            state1.dvar_M_HardwareMapDH_out_a_x2testing := TRUE;
            state1.dvar_M_HardwareMapDH := elit_init3;

            state0 := state1;
        END_IF;
    END_IF;

    // Event "tau".
    IF NOT progress THEN
        IF (state0.dvar_M_HardwareMapDH) = (elit_init3) THEN
            progress := TRUE;
            state1 := state0;

            state1.dvar_M_HardwareMapDH_out_a_transfer2pickpos := TRUE;
            state1.dvar_M_HardwareMapDH := elit_init4;

            state0 := state1;
        END_IF;
    END_IF;

    // Event "tau".
    IF NOT progress THEN
        b1 := (state0.dvar_M_HardwareMapDH) = (elit_init4);
        b1 := b1 AND (ivar_s_transfer_atpickup);
        IF b1 THEN
            progress := TRUE;
            state1 := state0;

            state1.dvar_M_HardwareMapDH_out_a_transfer2pickpos := FALSE;
            state1.dvar_M_HardwareMapDH := elit_init5;

            state0 := state1;
        END_IF;
    END_IF;

    // Event "tau".
    IF NOT progress THEN
        IF (state0.dvar_M_HardwareMapDH) = (elit_init5) THEN
            progress := TRUE;
            state1 := state0;

            state1.dvar_M_HardwareMapDH_out_a_transfer2droppos := TRUE;
            state1.dvar_M_HardwareMapDH := elit_init6;

            state0 := state1;
        END_IF;
    END_IF;

    // Event "tau".
    IF NOT progress THEN
        b1 := (state0.dvar_M_HardwareMapDH) = (elit_init6);
        b1 := b1 AND (ivar_s_transfer_athalfway);
        IF b1 THEN
            progress := TRUE;
            state1 := state0;

            state1.dvar_M_HardwareMapDH_out_a_transfer2droppos := FALSE;
            state1.dvar_M_HardwareMapDH := elit_init7;

            state0 := state1;
        END_IF;
    END_IF;

    // Event "tau".
    IF NOT progress THEN
        IF (state0.dvar_M_HardwareMapDH) = (elit_init7) THEN
            progress := TRUE;
            state1 := state0;

            state1.dvar_M_HardwareMapDH_out_a_x2distributing := FALSE;
            state1.dvar_M_HardwareMapDH := elit_init8;

            state0 := state1;
        END_IF;
    END_IF;

    // Event "tau".
    IF NOT progress THEN
        b1 := (state0.dvar_M_HardwareMapDH) = (elit_init8);
        b1 := b1 AND (ivar_s_xpos_atdrop);
        IF b1 THEN
            progress := TRUE;
            state1 := state0;

            state1.dvar_M_HardwareMapDH_out_a_x2distributing := TRUE;
            state1.cvar_M_HardwareMapDH_t := 0.0;
            state1.dvar_M_HardwareMapDH := elit_init9;

            state0 := state1;
        END_IF;
    END_IF;

    // Event "tau".
    IF NOT progress THEN
        b1 := (state0.dvar_M_HardwareMapDH) = (elit_init9);
        b1 := b1 AND ((state0.cvar_M_HardwareMapDH_t) >= (1));
        IF b1 THEN
            progress := TRUE;
            state1 := state0;

            state1.dvar_M_HardwareMapDH := elit_init_sensor_check;

            state0 := state1;
        END_IF;
    END_IF;

    // Event "tau".
    IF NOT progress THEN
        b1 := (state0.dvar_M_HardwareMapDH) = (elit_init_sensor_check);
        b1 := b1 AND (ivar_s_Dstartbutton);
        IF b1 THEN
            progress := TRUE;
            state1 := state0;

            state1.dvar_M_HardwareMapDH_init_err_sen_idx := 0;
            state1.dvar_M_HardwareMapDH := elit_init_error;

            state0 := state1;
        END_IF;
    END_IF;

    // Event "tau".
    IF NOT progress THEN
        b1 := (state0.dvar_M_HardwareMapDH) = (elit_init_sensor_check);
        b1 := b1 AND (NOT(ivar_s_Dstopbutton));
        IF b1 THEN
            progress := TRUE;
            state1 := state0;

            state1.dvar_M_HardwareMapDH_init_err_sen_idx := 1;
            state1.dvar_M_HardwareMapDH := elit_init_error;

            state0 := state1;
        END_IF;
    END_IF;

    // Event "tau".
    IF NOT progress THEN
        b1 := (state0.dvar_M_HardwareMapDH) = (elit_init_sensor_check);
        b1 := b1 AND (ivar_s_Dautoswitch);
        IF b1 THEN
            progress := TRUE;
            state1 := state0;

            state1.dvar_M_HardwareMapDH_init_err_sen_idx := 2;
            state1.dvar_M_HardwareMapDH := elit_init_error;

            state0 := state1;
        END_IF;
    END_IF;

    // Event "tau".
    IF NOT progress THEN
        b1 := (state0.dvar_M_HardwareMapDH) = (elit_init_sensor_check);
        b1 := b1 AND (ivar_s_Dresetbutton);
        IF b1 THEN
            progress := TRUE;
            state1 := state0;

            state1.dvar_M_HardwareMapDH_init_err_sen_idx := 3;
            state1.dvar_M_HardwareMapDH := elit_init_error;

            state0 := state1;
        END_IF;
    END_IF;

    // Event "tau".
    IF NOT progress THEN
        b1 := (state0.dvar_M_HardwareMapDH) = (elit_init_sensor_check);
        b1 := b1 AND (ivar_s_Din4);
        IF b1 THEN
            progress := TRUE;
            state1 := state0;

            state1.dvar_M_HardwareMapDH_init_err_sen_idx := 4;
            state1.dvar_M_HardwareMapDH := elit_init_error;

            state0 := state1;
        END_IF;
    END_IF;

    // Event "tau".
    IF NOT progress THEN
        b1 := (state0.dvar_M_HardwareMapDH) = (elit_init_sensor_check);
        b1 := b1 AND (ivar_s_Din5);
        IF b1 THEN
            progress := TRUE;
            state1 := state0;

            state1.dvar_M_HardwareMapDH_init_err_sen_idx := 5;
            state1.dvar_M_HardwareMapDH := elit_init_error;

            state0 := state1;
        END_IF;
    END_IF;

    // Event "tau".
    IF NOT progress THEN
        b1 := (state0.dvar_M_HardwareMapDH) = (elit_init_sensor_check);
        b1 := b1 AND (ivar_s_Din6);
        IF b1 THEN
            progress := TRUE;
            state1 := state0;

            state1.dvar_M_HardwareMapDH_init_err_sen_idx := 6;
            state1.dvar_M_HardwareMapDH := elit_init_error;

            state0 := state1;
        END_IF;
    END_IF;

    // Event "tau".
    IF NOT progress THEN
        b1 := (state0.dvar_M_HardwareMapDH) = (elit_init_sensor_check);
        b1 := b1 AND (ivar_s_Din7);
        IF b1 THEN
            progress := TRUE;
            state1 := state0;

            state1.dvar_M_HardwareMapDH_init_err_sen_idx := 7;
            state1.dvar_M_HardwareMapDH := elit_init_error;

            state0 := state1;
        END_IF;
    END_IF;

    // Event "tau".
    IF NOT progress THEN
        b1 := (state0.dvar_M_HardwareMapDH) = (elit_init_sensor_check);
        b1 := b1 AND (NOT(ivar_s_pusher1_in));
        IF b1 THEN
            progress := TRUE;
            state1 := state0;

            state1.dvar_M_HardwareMapDH_init_err_sen_idx := 8;
            state1.dvar_M_HardwareMapDH := elit_init_error;

            state0 := state1;
        END_IF;
    END_IF;

    // Event "tau".
    IF NOT progress THEN
        b1 := (state0.dvar_M_HardwareMapDH) = (elit_init_sensor_check);
        b1 := b1 AND (ivar_s_pusher1_out);
        IF b1 THEN
            progress := TRUE;
            state1 := state0;

            state1.dvar_M_HardwareMapDH_init_err_sen_idx := 9;
            state1.dvar_M_HardwareMapDH := elit_init_error;

            state0 := state1;
        END_IF;
    END_IF;

    // Event "tau".
    IF NOT progress THEN
        b1 := (state0.dvar_M_HardwareMapDH) = (elit_init_sensor_check);
        b1 := b1 AND (NOT(ivar_s_stack1filled));
        IF b1 THEN
            progress := TRUE;
            state1 := state0;

            state1.dvar_M_HardwareMapDH_init_err_sen_idx := 10;
            state1.dvar_M_HardwareMapDH := elit_init_error;

            state0 := state1;
        END_IF;
    END_IF;

    // Event "tau".
    IF NOT progress THEN
        b1 := (state0.dvar_M_HardwareMapDH) = (elit_init_sensor_check);
        b1 := b1 AND (ivar_s_product1);
        IF b1 THEN
            progress := TRUE;
            state1 := state0;

            state1.dvar_M_HardwareMapDH_init_err_sen_idx := 11;
            state1.dvar_M_HardwareMapDH := elit_init_error;

            state0 := state1;
        END_IF;
    END_IF;

    // Event "tau".
    IF NOT progress THEN
        b1 := (state0.dvar_M_HardwareMapDH) = (elit_init_sensor_check);
        b1 := b1 AND (NOT(ivar_s_pusher2_in));
        IF b1 THEN
            progress := TRUE;
            state1 := state0;

            state1.dvar_M_HardwareMapDH_init_err_sen_idx := 12;
            state1.dvar_M_HardwareMapDH := elit_init_error;

            state0 := state1;
        END_IF;
    END_IF;

    // Event "tau".
    IF NOT progress THEN
        b1 := (state0.dvar_M_HardwareMapDH) = (elit_init_sensor_check);
        b1 := b1 AND (ivar_s_pusher2_out);
        IF b1 THEN
            progress := TRUE;
            state1 := state0;

            state1.dvar_M_HardwareMapDH_init_err_sen_idx := 13;
            state1.dvar_M_HardwareMapDH := elit_init_error;

            state0 := state1;
        END_IF;
    END_IF;

    // Event "tau".
    IF NOT progress THEN
        b1 := (state0.dvar_M_HardwareMapDH) = (elit_init_sensor_check);
        b1 := b1 AND (NOT(ivar_s_stack2filled));
        IF b1 THEN
            progress := TRUE;
            state1 := state0;

            state1.dvar_M_HardwareMapDH_init_err_sen_idx := 14;
            state1.dvar_M_HardwareMapDH := elit_init_error;

            state0 := state1;
        END_IF;
    END_IF;

    // Event "tau".
    IF NOT progress THEN
        b1 := (state0.dvar_M_HardwareMapDH) = (elit_init_sensor_check);
        b1 := b1 AND (ivar_s_product2);
        IF b1 THEN
            progress := TRUE;
            state1 := state0;

            state1.dvar_M_HardwareMapDH_init_err_sen_idx := 15;
            state1.dvar_M_HardwareMapDH := elit_init_error;

            state0 := state1;
        END_IF;
    END_IF;

    // Event "tau".
    IF NOT progress THEN
        b1 := (state0.dvar_M_HardwareMapDH) = (elit_init_sensor_check);
        b1 := b1 AND (NOT(ivar_s_pusher3_in));
        IF b1 THEN
            progress := TRUE;
            state1 := state0;

            state1.dvar_M_HardwareMapDH_init_err_sen_idx := 16;
            state1.dvar_M_HardwareMapDH := elit_init_error;

            state0 := state1;
        END_IF;
    END_IF;

    // Event "tau".
    IF NOT progress THEN
        b1 := (state0.dvar_M_HardwareMapDH) = (elit_init_sensor_check);
        b1 := b1 AND (ivar_s_pusher3_out);
        IF b1 THEN
            progress := TRUE;
            state1 := state0;

            state1.dvar_M_HardwareMapDH_init_err_sen_idx := 17;
            state1.dvar_M_HardwareMapDH := elit_init_error;

            state0 := state1;
        END_IF;
    END_IF;

    // Event "tau".
    IF NOT progress THEN
        b1 := (state0.dvar_M_HardwareMapDH) = (elit_init_sensor_check);
        b1 := b1 AND (NOT(ivar_s_stack3filled));
        IF b1 THEN
            progress := TRUE;
            state1 := state0;

            state1.dvar_M_HardwareMapDH_init_err_sen_idx := 18;
            state1.dvar_M_HardwareMapDH := elit_init_error;

            state0 := state1;
        END_IF;
    END_IF;

    // Event "tau".
    IF NOT progress THEN
        b1 := (state0.dvar_M_HardwareMapDH) = (elit_init_sensor_check);
        b1 := b1 AND (ivar_s_product3);
        IF b1 THEN
            progress := TRUE;
            state1 := state0;

            state1.dvar_M_HardwareMapDH_init_err_sen_idx := 19;
            state1.dvar_M_HardwareMapDH := elit_init_error;

            state0 := state1;
        END_IF;
    END_IF;

    // Event "tau".
    IF NOT progress THEN
        b1 := (state0.dvar_M_HardwareMapDH) = (elit_init_sensor_check);
        b1 := b1 AND (ivar_s_Hstartbutton);
        IF b1 THEN
            progress := TRUE;
            state1 := state0;

            state1.dvar_M_HardwareMapDH_init_err_sen_idx := 22;
            state1.dvar_M_HardwareMapDH := elit_init_error;

            state0 := state1;
        END_IF;
    END_IF;

    // Event "tau".
    IF NOT progress THEN
        b1 := (state0.dvar_M_HardwareMapDH) = (elit_init_sensor_check);
        b1 := b1 AND (NOT(ivar_s_Hstopbutton));
        IF b1 THEN
            progress := TRUE;
            state1 := state0;

            state1.dvar_M_HardwareMapDH_init_err_sen_idx := 23;
            state1.dvar_M_HardwareMapDH := elit_init_error;

            state0 := state1;
        END_IF;
    END_IF;

    // Event "tau".
    IF NOT progress THEN
        b1 := (state0.dvar_M_HardwareMapDH) = (elit_init_sensor_check);
        b1 := b1 AND (ivar_s_Hautoswitch);
        IF b1 THEN
            progress := TRUE;
            state1 := state0;

            state1.dvar_M_HardwareMapDH_init_err_sen_idx := 24;
            state1.dvar_M_HardwareMapDH := elit_init_error;

            state0 := state1;
        END_IF;
    END_IF;

    // Event "tau".
    IF NOT progress THEN
        b1 := (state0.dvar_M_HardwareMapDH) = (elit_init_sensor_check);
        b1 := b1 AND (ivar_s_Hresetbutton);
        IF b1 THEN
            progress := TRUE;
            state1 := state0;

            state1.dvar_M_HardwareMapDH_init_err_sen_idx := 25;
            state1.dvar_M_HardwareMapDH := elit_init_error;

            state0 := state1;
        END_IF;
    END_IF;

    // Event "tau".
    IF NOT progress THEN
        b1 := (state0.dvar_M_HardwareMapDH) = (elit_init_sensor_check);
        b1 := b1 AND (ivar_s_Hin4);
        IF b1 THEN
            progress := TRUE;
            state1 := state0;

            state1.dvar_M_HardwareMapDH_init_err_sen_idx := 26;
            state1.dvar_M_HardwareMapDH := elit_init_error;

            state0 := state1;
        END_IF;
    END_IF;

    // Event "tau".
    IF NOT progress THEN
        b1 := (state0.dvar_M_HardwareMapDH) = (elit_init_sensor_check);
        b1 := b1 AND (ivar_s_Hin5);
        IF b1 THEN
            progress := TRUE;
            state1 := state0;

            state1.dvar_M_HardwareMapDH_init_err_sen_idx := 27;
            state1.dvar_M_HardwareMapDH := elit_init_error;

            state0 := state1;
        END_IF;
    END_IF;

    // Event "tau".
    IF NOT progress THEN
        b1 := (state0.dvar_M_HardwareMapDH) = (elit_init_sensor_check);
        b1 := b1 AND (ivar_s_Hin6);
        IF b1 THEN
            progress := TRUE;
            state1 := state0;

            state1.dvar_M_HardwareMapDH_init_err_sen_idx := 28;
            state1.dvar_M_HardwareMapDH := elit_init_error;

            state0 := state1;
        END_IF;
    END_IF;

    // Event "tau".
    IF NOT progress THEN
        b1 := (state0.dvar_M_HardwareMapDH) = (elit_init_sensor_check);
        b1 := b1 AND (ivar_s_Hin7);
        IF b1 THEN
            progress := TRUE;
            state1 := state0;

            state1.dvar_M_HardwareMapDH_init_err_sen_idx := 29;
            state1.dvar_M_HardwareMapDH := elit_init_error;

            state0 := state1;
        END_IF;
    END_IF;

    // Event "tau".
    IF NOT progress THEN
        b1 := (state0.dvar_M_HardwareMapDH) = (elit_init_sensor_check);
        b1 := b1 AND (ivar_s_xpos_at1);
        IF b1 THEN
            progress := TRUE;
            state1 := state0;

            state1.dvar_M_HardwareMapDH_init_err_sen_idx := 33;
            state1.dvar_M_HardwareMapDH := elit_init_error;

            state0 := state1;
        END_IF;
    END_IF;

    // Event "tau".
    IF NOT progress THEN
        b1 := (state0.dvar_M_HardwareMapDH) = (elit_init_sensor_check);
        b1 := b1 AND (ivar_s_xpos_at2);
        IF b1 THEN
            progress := TRUE;
            state1 := state0;

            state1.dvar_M_HardwareMapDH_init_err_sen_idx := 34;
            state1.dvar_M_HardwareMapDH := elit_init_error;

            state0 := state1;
        END_IF;
    END_IF;

    // Event "tau".
    IF NOT progress THEN
        b1 := (state0.dvar_M_HardwareMapDH) = (elit_init_sensor_check);
        b1 := b1 AND (ivar_s_xpos_at3);
        IF b1 THEN
            progress := TRUE;
            state1 := state0;

            state1.dvar_M_HardwareMapDH_init_err_sen_idx := 35;
            state1.dvar_M_HardwareMapDH := elit_init_error;

            state0 := state1;
        END_IF;
    END_IF;

    // Event "tau".
    IF NOT progress THEN
        b1 := (state0.dvar_M_HardwareMapDH) = (elit_init_sensor_check);
        b1 := b1 AND (NOT(ivar_s_xpos_atdrop));
        IF b1 THEN
            progress := TRUE;
            state1 := state0;

            state1.dvar_M_HardwareMapDH_init_err_sen_idx := 36;
            state1.dvar_M_HardwareMapDH := elit_init_error;

            state0 := state1;
        END_IF;
    END_IF;

    // Event "tau".
    IF NOT progress THEN
        b1 := (state0.dvar_M_HardwareMapDH) = (elit_init_sensor_check);
        b1 := b1 AND (NOT(ivar_s_zpos_atup));
        IF b1 THEN
            progress := TRUE;
            state1 := state0;

            state1.dvar_M_HardwareMapDH_init_err_sen_idx := 37;
            state1.dvar_M_HardwareMapDH := elit_init_error;

            state0 := state1;
        END_IF;
    END_IF;

    // Event "tau".
    IF NOT progress THEN
        b1 := (state0.dvar_M_HardwareMapDH) = (elit_init_sensor_check);
        b1 := b1 AND (ivar_s_zpos_atdown);
        IF b1 THEN
            progress := TRUE;
            state1 := state0;

            state1.dvar_M_HardwareMapDH_init_err_sen_idx := 38;
            state1.dvar_M_HardwareMapDH := elit_init_error;

            state0 := state1;
        END_IF;
    END_IF;

    // Event "tau".
    IF NOT progress THEN
        b1 := (state0.dvar_M_HardwareMapDH) = (elit_init_sensor_check);
        b1 := b1 AND (ivar_s_gripper);
        IF b1 THEN
            progress := TRUE;
            state1 := state0;

            state1.dvar_M_HardwareMapDH_init_err_sen_idx := 39;
            state1.dvar_M_HardwareMapDH := elit_init_error;

            state0 := state1;
        END_IF;
    END_IF;

    // Event "tau".
    IF NOT progress THEN
        b1 := (state0.dvar_M_HardwareMapDH) = (elit_init_sensor_check);
        b1 := b1 AND (ivar_s_transfer_atpickup);
        IF b1 THEN
            progress := TRUE;
            state1 := state0;

            state1.dvar_M_HardwareMapDH_init_err_sen_idx := 40;
            state1.dvar_M_HardwareMapDH := elit_init_error;

            state0 := state1;
        END_IF;
    END_IF;

    // Event "tau".
    IF NOT progress THEN
        b1 := (state0.dvar_M_HardwareMapDH) = (elit_init_sensor_check);
        b1 := b1 AND (ivar_s_transfer_atdrop);
        IF b1 THEN
            progress := TRUE;
            state1 := state0;

            state1.dvar_M_HardwareMapDH_init_err_sen_idx := 41;
            state1.dvar_M_HardwareMapDH := elit_init_error;

            state0 := state1;
        END_IF;
    END_IF;

    // Event "tau".
    IF NOT progress THEN
        b1 := (state0.dvar_M_HardwareMapDH) = (elit_init_sensor_check);
        b1 := b1 AND (NOT(ivar_s_transfer_athalfway));
        IF b1 THEN
            progress := TRUE;
            state1 := state0;

            state1.dvar_M_HardwareMapDH_init_err_sen_idx := 42;
            state1.dvar_M_HardwareMapDH := elit_init_error;

            state0 := state1;
        END_IF;
    END_IF;

    // Event "tau".
    IF NOT progress THEN
        b1 := (state0.dvar_M_HardwareMapDH) = (elit_init_sensor_check);
        b1 := b1 AND (ivar_s_vacuum);
        IF b1 THEN
            progress := TRUE;
            state1 := state0;

            state1.dvar_M_HardwareMapDH_init_err_sen_idx := 43;
            state1.dvar_M_HardwareMapDH := elit_init_error;

            state0 := state1;
        END_IF;
    END_IF;

    // Event "tau".
    IF NOT progress THEN
        b1 := (state0.dvar_M_HardwareMapDH) = (elit_init_sensor_check);
        b1 := b1 AND (ivar_s_product4);
        IF b1 THEN
            progress := TRUE;
            state1 := state0;

            state1.dvar_M_HardwareMapDH_init_err_sen_idx := 44;
            state1.dvar_M_HardwareMapDH := elit_init_error;

            state0 := state1;
        END_IF;
    END_IF;

    // Event "tau".
    IF NOT progress THEN
        b1 := (state0.dvar_M_HardwareMapDH) = (elit_init_sensor_check);
        b1 := b1 AND (NOT(ivar_s_Dstartbutton));
        b1 := b1 AND (ivar_s_Dstopbutton);
        b1 := b1 AND (NOT(ivar_s_Dautoswitch));
        b1 := b1 AND (NOT(ivar_s_Dresetbutton));
        b1 := b1 AND (NOT(ivar_s_Din4));
        b1 := b1 AND (NOT(ivar_s_Din5));
        b1 := b1 AND (NOT(ivar_s_Din6));
        b1 := b1 AND (NOT(ivar_s_Din7));
        b1 := b1 AND (ivar_s_pusher1_in);
        b1 := b1 AND (NOT(ivar_s_pusher1_out));
        b1 := b1 AND (ivar_s_stack1filled);
        b1 := b1 AND (NOT(ivar_s_product1));
        b1 := b1 AND (ivar_s_pusher2_in);
        b1 := b1 AND (NOT(ivar_s_pusher2_out));
        b1 := b1 AND (ivar_s_stack2filled);
        b1 := b1 AND (NOT(ivar_s_product2));
        b1 := b1 AND (ivar_s_pusher3_in);
        b1 := b1 AND (NOT(ivar_s_pusher3_out));
        b1 := b1 AND (ivar_s_stack3filled);
        b1 := b1 AND (NOT(ivar_s_product3));
        b1 := b1 AND (NOT(ivar_s_Hstartbutton));
        b1 := b1 AND (ivar_s_Hstopbutton);
        b1 := b1 AND (NOT(ivar_s_Hautoswitch));
        b1 := b1 AND (NOT(ivar_s_Hresetbutton));
        b1 := b1 AND (NOT(ivar_s_Hin4));
        b1 := b1 AND (NOT(ivar_s_Hin5));
        b1 := b1 AND (NOT(ivar_s_Hin6));
        b1 := b1 AND (NOT(ivar_s_Hin7));
        b1 := b1 AND (NOT(ivar_s_xpos_at1));
        b1 := b1 AND (NOT(ivar_s_xpos_at2));
        b1 := b1 AND (NOT(ivar_s_xpos_at3));
        b1 := b1 AND (ivar_s_xpos_atdrop);
        b1 := b1 AND (ivar_s_zpos_atup);
        b1 := b1 AND (NOT(ivar_s_zpos_atdown));
        b1 := b1 AND (NOT(ivar_s_gripper));
        b1 := b1 AND (NOT(ivar_s_transfer_atpickup));
        b1 := b1 AND (NOT(ivar_s_transfer_atdrop));
        b1 := b1 AND (ivar_s_transfer_athalfway);
        b1 := b1 AND (NOT(ivar_s_vacuum));
        b1 := b1 AND (NOT(ivar_s_product4));
        IF b1 THEN
            progress := TRUE;
            state1 := state0;

            state1.dvar_M_HardwareMapDH := elit_init_ok;

            state0 := state1;
        END_IF;
    END_IF;

    // Event "tau".
    IF NOT progress THEN
        b1 := (state0.dvar_M_HardwareMapDH) = (elit_init_error);
        b1 := b1 AND ((state0.cvar_M_HardwareMapDH_t) >= (0.5));
        b1 := b1 AND ((state0.dvar_M_HardwareMapDH_init_err_led_idx) = (0));
        IF b1 THEN
            progress := TRUE;
            state1 := state0;

            state1.cvar_M_HardwareMapDH_t := 0.0;
            state1.dvar_M_HardwareMapDH_init_err_led_idx := 1;
            state1.dvar_M_HardwareMapDH_out_a_DledQ1 := TRUE;
            state1.dvar_M_HardwareMapDH_out_a_DledQ2 := FALSE;
            state1.dvar_M_HardwareMapDH_out_a_HledQ1 := TRUE;
            state1.dvar_M_HardwareMapDH_out_a_HledQ2 := FALSE;

            state0 := state1;
        END_IF;
    END_IF;

    // Event "tau".
    IF NOT progress THEN
        b1 := (state0.dvar_M_HardwareMapDH) = (elit_init_error);
        b1 := b1 AND ((state0.cvar_M_HardwareMapDH_t) >= (0.5));
        b1 := b1 AND ((state0.dvar_M_HardwareMapDH_init_err_led_idx) = (1));
        IF b1 THEN
            progress := TRUE;
            state1 := state0;

            state1.cvar_M_HardwareMapDH_t := 0.0;
            state1.dvar_M_HardwareMapDH_init_err_led_idx := 0;
            state1.dvar_M_HardwareMapDH_out_a_DledQ1 := FALSE;
            state1.dvar_M_HardwareMapDH_out_a_DledQ2 := TRUE;
            state1.dvar_M_HardwareMapDH_out_a_HledQ1 := FALSE;
            state1.dvar_M_HardwareMapDH_out_a_HledQ2 := TRUE;

            state0 := state1;
        END_IF;
    END_IF;

    // Event "tau".
    IF NOT progress THEN
        IF (state0.dvar_M_HardwareMapDH) = (elit_init_ok) THEN
            progress := TRUE;
            state1 := state0;

            state1.dvar_M_HardwareMapDH_out_a_DledQ1 := FALSE;
            state1.dvar_M_HardwareMapDH_out_a_DledQ2 := FALSE;
            state1.dvar_M_HardwareMapDH_out_a_HledQ1 := FALSE;
            state1.dvar_M_HardwareMapDH_out_a_HledQ2 := FALSE;
            state1.dvar_M_HardwareMapDH := elit_initialized;

            state0 := state1;
        END_IF;
    END_IF;

    // Event "tau".
    IF NOT progress THEN
        b1 := (state0.dvar_M_HardwareMapDH) = (elit_initialized);
        b1 := b1 AND ((state0.dvar_M_HardwareMapDH_out_a_Dstartled) <> (FALSE));
        IF b1 THEN
            progress := TRUE;
            state1 := state0;

            state1.dvar_M_HardwareMapDH_out_a_Dstartled := FALSE;

            state0 := state1;
        END_IF;
    END_IF;

    // Event "tau".
    IF NOT progress THEN
        b1 := (state0.dvar_M_HardwareMapDH) = (elit_initialized);
        b1 := b1 AND ((state0.dvar_M_HardwareMapDH_out_a_Dresetled) <> (FALSE));
        IF b1 THEN
            progress := TRUE;
            state1 := state0;

            state1.dvar_M_HardwareMapDH_out_a_Dresetled := FALSE;

            state0 := state1;
        END_IF;
    END_IF;

    // Event "tau".
    IF NOT progress THEN
        b1 := (state0.dvar_M_HardwareMapDH) = (elit_initialized);
        b1 := b1 AND ((state0.dvar_M_HardwareMapDH_out_a_DledQ1) <> (FALSE));
        IF b1 THEN
            progress := TRUE;
            state1 := state0;

            state1.dvar_M_HardwareMapDH_out_a_DledQ1 := FALSE;

            state0 := state1;
        END_IF;
    END_IF;

    // Event "tau".
    IF NOT progress THEN
        b1 := (state0.dvar_M_HardwareMapDH) = (elit_initialized);
        b1 := b1 AND ((state0.dvar_M_HardwareMapDH_out_a_DledQ2) <> (FALSE));
        IF b1 THEN
            progress := TRUE;
            state1 := state0;

            state1.dvar_M_HardwareMapDH_out_a_DledQ2 := FALSE;

            state0 := state1;
        END_IF;
    END_IF;

    // Event "tau".
    IF NOT progress THEN
        b1 := (state0.dvar_M_HardwareMapDH) = (elit_initialized);
        b1 := b1 AND ((state0.dvar_M_HardwareMapDH_out_a_Dout4) <> (FALSE));
        IF b1 THEN
            progress := TRUE;
            state1 := state0;

            state1.dvar_M_HardwareMapDH_out_a_Dout4 := FALSE;

            state0 := state1;
        END_IF;
    END_IF;

    // Event "tau".
    IF NOT progress THEN
        b1 := (state0.dvar_M_HardwareMapDH) = (elit_initialized);
        b1 := b1 AND ((state0.dvar_M_HardwareMapDH_out_a_Dout5) <> (FALSE));
        IF b1 THEN
            progress := TRUE;
            state1 := state0;

            state1.dvar_M_HardwareMapDH_out_a_Dout5 := FALSE;

            state0 := state1;
        END_IF;
    END_IF;

    // Event "tau".
    IF NOT progress THEN
        b1 := (state0.dvar_M_HardwareMapDH) = (elit_initialized);
        b1 := b1 AND ((state0.dvar_M_HardwareMapDH_out_a_Dout6) <> (FALSE));
        IF b1 THEN
            progress := TRUE;
            state1 := state0;

            state1.dvar_M_HardwareMapDH_out_a_Dout6 := FALSE;

            state0 := state1;
        END_IF;
    END_IF;

    // Event "tau".
    IF NOT progress THEN
        b1 := (state0.dvar_M_HardwareMapDH) = (elit_initialized);
        b1 := b1 AND ((state0.dvar_M_HardwareMapDH_out_a_Dout7) <> (FALSE));
        IF b1 THEN
            progress := TRUE;
            state1 := state0;

            state1.dvar_M_HardwareMapDH_out_a_Dout7 := FALSE;

            state0 := state1;
        END_IF;
    END_IF;

    // Event "tau".
    IF NOT progress THEN
        b1 := (state0.dvar_M_HardwareMapDH) = (elit_initialized);
        b1 := b1 AND ((state0.dvar_M_HardwareMapDH_out_a_pusher1) <> ((state0.dvar_M_sup_A_pusher1) = (elit_On)));
        IF b1 THEN
            progress := TRUE;
            state1 := state0;

            state1.dvar_M_HardwareMapDH_out_a_pusher1 := (state0.dvar_M_sup_A_pusher1) = (elit_On);

            state0 := state1;
        END_IF;
    END_IF;

    // Event "tau".
    IF NOT progress THEN
        b1 := (state0.dvar_M_HardwareMapDH) = (elit_initialized);
        b1 := b1 AND ((state0.dvar_M_HardwareMapDH_out_a_pusher2) <> ((state0.dvar_M_sup_A_pusher2) = (elit_On)));
        IF b1 THEN
            progress := TRUE;
            state1 := state0;

            state1.dvar_M_HardwareMapDH_out_a_pusher2 := (state0.dvar_M_sup_A_pusher2) = (elit_On);

            state0 := state1;
        END_IF;
    END_IF;

    // Event "tau".
    IF NOT progress THEN
        b1 := (state0.dvar_M_HardwareMapDH) = (elit_initialized);
        b1 := b1 AND ((state0.dvar_M_HardwareMapDH_out_a_pusher3) <> ((state0.dvar_M_sup_A_pusher3) = (elit_On)));
        IF b1 THEN
            progress := TRUE;
            state1 := state0;

            state1.dvar_M_HardwareMapDH_out_a_pusher3 := (state0.dvar_M_sup_A_pusher3) = (elit_On);

            state0 := state1;
        END_IF;
    END_IF;

    // Event "tau".
    IF NOT progress THEN
        b1 := (state0.dvar_M_HardwareMapDH) = (elit_initialized);
        b1 := b1 AND ((state0.dvar_M_HardwareMapDH_out_a_Hstartled) <> (FALSE));
        IF b1 THEN
            progress := TRUE;
            state1 := state0;

            state1.dvar_M_HardwareMapDH_out_a_Hstartled := FALSE;

            state0 := state1;
        END_IF;
    END_IF;

    // Event "tau".
    IF NOT progress THEN
        b1 := (state0.dvar_M_HardwareMapDH) = (elit_initialized);
        b1 := b1 AND ((state0.dvar_M_HardwareMapDH_out_a_Hresetled) <> (FALSE));
        IF b1 THEN
            progress := TRUE;
            state1 := state0;

            state1.dvar_M_HardwareMapDH_out_a_Hresetled := FALSE;

            state0 := state1;
        END_IF;
    END_IF;

    // Event "tau".
    IF NOT progress THEN
        b1 := (state0.dvar_M_HardwareMapDH) = (elit_initialized);
        b1 := b1 AND ((state0.dvar_M_HardwareMapDH_out_a_HledQ1) <> (FALSE));
        IF b1 THEN
            progress := TRUE;
            state1 := state0;

            state1.dvar_M_HardwareMapDH_out_a_HledQ1 := FALSE;

            state0 := state1;
        END_IF;
    END_IF;

    // Event "tau".
    IF NOT progress THEN
        b1 := (state0.dvar_M_HardwareMapDH) = (elit_initialized);
        b1 := b1 AND ((state0.dvar_M_HardwareMapDH_out_a_HledQ2) <> (FALSE));
        IF b1 THEN
            progress := TRUE;
            state1 := state0;

            state1.dvar_M_HardwareMapDH_out_a_HledQ2 := FALSE;

            state0 := state1;
        END_IF;
    END_IF;

    // Event "tau".
    IF NOT progress THEN
        b1 := (state0.dvar_M_HardwareMapDH) = (elit_initialized);
        b1 := b1 AND ((state0.dvar_M_HardwareMapDH_out_a_Hout4) <> (FALSE));
        IF b1 THEN
            progress := TRUE;
            state1 := state0;

            state1.dvar_M_HardwareMapDH_out_a_Hout4 := FALSE;

            state0 := state1;
        END_IF;
    END_IF;

    // Event "tau".
    IF NOT progress THEN
        b1 := (state0.dvar_M_HardwareMapDH) = (elit_initialized);
        b1 := b1 AND ((state0.dvar_M_HardwareMapDH_out_a_Hout5) <> (FALSE));
        IF b1 THEN
            progress := TRUE;
            state1 := state0;

            state1.dvar_M_HardwareMapDH_out_a_Hout5 := FALSE;

            state0 := state1;
        END_IF;
    END_IF;

    // Event "tau".
    IF NOT progress THEN
        b1 := (state0.dvar_M_HardwareMapDH) = (elit_initialized);
        b1 := b1 AND ((state0.dvar_M_HardwareMapDH_out_a_Hout6) <> (FALSE));
        IF b1 THEN
            progress := TRUE;
            state1 := state0;

            state1.dvar_M_HardwareMapDH_out_a_Hout6 := FALSE;

            state0 := state1;
        END_IF;
    END_IF;

    // Event "tau".
    IF NOT progress THEN
        b1 := (state0.dvar_M_HardwareMapDH) = (elit_initialized);
        b1 := b1 AND ((state0.dvar_M_HardwareMapDH_out_a_Hout7) <> (FALSE));
        IF b1 THEN
            progress := TRUE;
            state1 := state0;

            state1.dvar_M_HardwareMapDH_out_a_Hout7 := FALSE;

            state0 := state1;
        END_IF;
    END_IF;

    // Event "tau".
    IF NOT progress THEN
        b1 := (state0.dvar_M_HardwareMapDH) = (elit_initialized);
        b1 := b1 AND ((state0.dvar_M_HardwareMapDH_out_a_x2distributing) <> ((state0.dvar_M_sup_A_x2distributing) = (elit_On)));
        IF b1 THEN
            progress := TRUE;
            state1 := state0;

            state1.dvar_M_HardwareMapDH_out_a_x2distributing := (state0.dvar_M_sup_A_x2distributing) = (elit_On);

            state0 := state1;
        END_IF;
    END_IF;

    // Event "tau".
    IF NOT progress THEN
        b1 := (state0.dvar_M_HardwareMapDH) = (elit_initialized);
        b1 := b1 AND ((state0.dvar_M_HardwareMapDH_out_a_x2testing) <> ((state0.dvar_M_sup_A_x2testing) = (elit_On)));
        IF b1 THEN
            progress := TRUE;
            state1 := state0;

            state1.dvar_M_HardwareMapDH_out_a_x2testing := (state0.dvar_M_sup_A_x2testing) = (elit_On);

            state0 := state1;
        END_IF;
    END_IF;

    // Event "tau".
    IF NOT progress THEN
        b1 := (state0.dvar_M_HardwareMapDH) = (elit_initialized);
        b1 := b1 AND ((state0.dvar_M_HardwareMapDH_out_a_zdown) <> ((state0.dvar_M_sup_A_zdown) = (elit_On)));
        IF b1 THEN
            progress := TRUE;
            state1 := state0;

            state1.dvar_M_HardwareMapDH_out_a_zdown := (state0.dvar_M_sup_A_zdown) = (elit_On);

            state0 := state1;
        END_IF;
    END_IF;

    // Event "tau".
    IF NOT progress THEN
        b1 := (state0.dvar_M_HardwareMapDH) = (elit_initialized);
        b1 := b1 AND ((state0.dvar_M_HardwareMapDH_out_a_gripperclose) <> ((state0.dvar_M_sup_A_gripperclose) = (elit_On)));
        IF b1 THEN
            progress := TRUE;
            state1 := state0;

            state1.dvar_M_HardwareMapDH_out_a_gripperclose := (state0.dvar_M_sup_A_gripperclose) = (elit_On);

            state0 := state1;
        END_IF;
    END_IF;

    // Event "tau".
    IF NOT progress THEN
        b1 := (state0.dvar_M_HardwareMapDH) = (elit_initialized);
        b1 := b1 AND ((state0.dvar_M_HardwareMapDH_out_a_transfer2pickpos) <> ((state0.dvar_M_sup_A_transfer2pickpos) = (elit_On)));
        IF b1 THEN
            progress := TRUE;
            state1 := state0;

            state1.dvar_M_HardwareMapDH_out_a_transfer2pickpos := (state0.dvar_M_sup_A_transfer2pickpos) = (elit_On);

            state0 := state1;
        END_IF;
    END_IF;

    // Event "tau".
    IF NOT progress THEN
        b1 := (state0.dvar_M_HardwareMapDH) = (elit_initialized);
        b1 := b1 AND ((state0.dvar_M_HardwareMapDH_out_a_transfer2droppos) <> ((state0.dvar_M_sup_A_transfer2droppos) = (elit_On)));
        IF b1 THEN
            progress := TRUE;
            state1 := state0;

            state1.dvar_M_HardwareMapDH_out_a_transfer2droppos := (state0.dvar_M_sup_A_transfer2droppos) = (elit_On);

            state0 := state1;
        END_IF;
    END_IF;

    // Event "tau".
    IF NOT progress THEN
        b1 := (state0.dvar_M_HardwareMapDH) = (elit_initialized);
        b1 := b1 AND ((state0.dvar_M_HardwareMapDH_out_a_vacuum) <> ((state0.dvar_M_sup_A_vacuum) = (elit_On)));
        IF b1 THEN
            progress := TRUE;
            state1 := state0;

            state1.dvar_M_HardwareMapDH_out_a_vacuum := (state0.dvar_M_sup_A_vacuum) = (elit_On);

            state0 := state1;
        END_IF;
    END_IF;

    // Event "tau".
    IF NOT progress THEN
        b1 := (state0.dvar_M_HardwareMapDH) = (elit_initialized);
        b1 := b1 AND ((state0.dvar_M_HardwareMapDH_out_a_ejectpulse) <> ((state0.dvar_M_sup_A_ejectpulse) = (elit_On)));
        IF b1 THEN
            progress := TRUE;
            state1 := state0;

            state1.dvar_M_HardwareMapDH_out_a_ejectpulse := (state0.dvar_M_sup_A_ejectpulse) = (elit_On);

            state0 := state1;
        END_IF;
    END_IF;

    // Event "tau".
    IF NOT progress THEN
        b1 := (state0.dvar_M_HardwareMapDH) = (elit_initialized);
        b1 := b1 AND ((state0.dvar_M_HardwareMapDH_out_a_handlingready) <> ((state0.dvar_M_sup_A_handlingready) = (elit_On)));
        IF b1 THEN
            progress := TRUE;
            state1 := state0;

            state1.dvar_M_HardwareMapDH_out_a_handlingready := (state0.dvar_M_sup_A_handlingready) = (elit_On);

            state0 := state1;
        END_IF;
    END_IF;

    // Event "tau".
    IF NOT progress THEN
        b1 := (state0.dvar_M_HardwareMapP) = (elit_init0);
        b1 := b1 AND ((state0.cvar_M_HardwareMapP_t) >= (2.0));
        IF b1 THEN
            progress := TRUE;
            state1 := state0;

            state1.dvar_M_HardwareMapP := elit_init1;

            state0 := state1;
        END_IF;
    END_IF;

    // Event "tau".
    IF NOT progress THEN
        IF (state0.dvar_M_HardwareMapP) = (elit_init1) THEN
            progress := TRUE;
            state1 := state0;

            state1.dvar_M_HardwareMapP_out_a_turntable := TRUE;
            state1.dvar_M_HardwareMapP := elit_init2;

            state0 := state1;
        END_IF;
    END_IF;

    // Event "tau".
    IF NOT progress THEN
        b1 := (state0.dvar_M_HardwareMapP) = (elit_init2);
        b1 := b1 AND (NOT(ivar_s_turntable));
        IF b1 THEN
            progress := TRUE;
            state1 := state0;

            state1.dvar_M_HardwareMapP := elit_init3;

            state0 := state1;
        END_IF;
    END_IF;

    // Event "tau".
    IF NOT progress THEN
        b1 := (state0.dvar_M_HardwareMapP) = (elit_init3);
        b1 := b1 AND (ivar_s_turntable);
        IF b1 THEN
            progress := TRUE;
            state1 := state0;

            state1.dvar_M_HardwareMapP_out_a_turntable := FALSE;
            state1.cvar_M_HardwareMapP_t := 0.0;
            state1.dvar_M_HardwareMapP := elit_init4;

            state0 := state1;
        END_IF;
    END_IF;

    // Event "tau".
    IF NOT progress THEN
        b1 := (state0.dvar_M_HardwareMapP) = (elit_init4);
        b1 := b1 AND ((state0.cvar_M_HardwareMapP_t) >= (1));
        IF b1 THEN
            progress := TRUE;
            state1 := state0;

            state1.dvar_M_HardwareMapP := elit_init_sensor_check;

            state0 := state1;
        END_IF;
    END_IF;

    // Event "tau".
    IF NOT progress THEN
        b1 := (state0.dvar_M_HardwareMapP) = (elit_init_sensor_check);
        b1 := b1 AND (ivar_s_Pstartbutton);
        IF b1 THEN
            progress := TRUE;
            state1 := state0;

            state1.dvar_M_HardwareMapP_init_err_sen_idx := 0;
            state1.dvar_M_HardwareMapP := elit_init_error;

            state0 := state1;
        END_IF;
    END_IF;

    // Event "tau".
    IF NOT progress THEN
        b1 := (state0.dvar_M_HardwareMapP) = (elit_init_sensor_check);
        b1 := b1 AND (NOT(ivar_s_Pstopbutton));
        IF b1 THEN
            progress := TRUE;
            state1 := state0;

            state1.dvar_M_HardwareMapP_init_err_sen_idx := 1;
            state1.dvar_M_HardwareMapP := elit_init_error;

            state0 := state1;
        END_IF;
    END_IF;

    // Event "tau".
    IF NOT progress THEN
        b1 := (state0.dvar_M_HardwareMapP) = (elit_init_sensor_check);
        b1 := b1 AND (ivar_s_Pautoswitch);
        IF b1 THEN
            progress := TRUE;
            state1 := state0;

            state1.dvar_M_HardwareMapP_init_err_sen_idx := 2;
            state1.dvar_M_HardwareMapP := elit_init_error;

            state0 := state1;
        END_IF;
    END_IF;

    // Event "tau".
    IF NOT progress THEN
        b1 := (state0.dvar_M_HardwareMapP) = (elit_init_sensor_check);
        b1 := b1 AND (ivar_s_Presetbutton);
        IF b1 THEN
            progress := TRUE;
            state1 := state0;

            state1.dvar_M_HardwareMapP_init_err_sen_idx := 3;
            state1.dvar_M_HardwareMapP := elit_init_error;

            state0 := state1;
        END_IF;
    END_IF;

    // Event "tau".
    IF NOT progress THEN
        b1 := (state0.dvar_M_HardwareMapP) = (elit_init_sensor_check);
        b1 := b1 AND (ivar_s_Pin4);
        IF b1 THEN
            progress := TRUE;
            state1 := state0;

            state1.dvar_M_HardwareMapP_init_err_sen_idx := 4;
            state1.dvar_M_HardwareMapP := elit_init_error;

            state0 := state1;
        END_IF;
    END_IF;

    // Event "tau".
    IF NOT progress THEN
        b1 := (state0.dvar_M_HardwareMapP) = (elit_init_sensor_check);
        b1 := b1 AND (ivar_s_Pin5);
        IF b1 THEN
            progress := TRUE;
            state1 := state0;

            state1.dvar_M_HardwareMapP_init_err_sen_idx := 5;
            state1.dvar_M_HardwareMapP := elit_init_error;

            state0 := state1;
        END_IF;
    END_IF;

    // Event "tau".
    IF NOT progress THEN
        b1 := (state0.dvar_M_HardwareMapP) = (elit_init_sensor_check);
        b1 := b1 AND (ivar_s_Pin6);
        IF b1 THEN
            progress := TRUE;
            state1 := state0;

            state1.dvar_M_HardwareMapP_init_err_sen_idx := 6;
            state1.dvar_M_HardwareMapP := elit_init_error;

            state0 := state1;
        END_IF;
    END_IF;

    // Event "tau".
    IF NOT progress THEN
        b1 := (state0.dvar_M_HardwareMapP) = (elit_init_sensor_check);
        b1 := b1 AND (ivar_s_Pin7);
        IF b1 THEN
            progress := TRUE;
            state1 := state0;

            state1.dvar_M_HardwareMapP_init_err_sen_idx := 7;
            state1.dvar_M_HardwareMapP := elit_init_error;

            state0 := state1;
        END_IF;
    END_IF;

    // Event "tau".
    IF NOT progress THEN
        b1 := (state0.dvar_M_HardwareMapP) = (elit_init_sensor_check);
        b1 := b1 AND (ivar_s_atinput);
        IF b1 THEN
            progress := TRUE;
            state1 := state0;

            state1.dvar_M_HardwareMapP_init_err_sen_idx := 8;
            state1.dvar_M_HardwareMapP := elit_init_error;

            state0 := state1;
        END_IF;
    END_IF;

    // Event "tau".
    IF NOT progress THEN
        b1 := (state0.dvar_M_HardwareMapP) = (elit_init_sensor_check);
        b1 := b1 AND (ivar_s_attest);
        IF b1 THEN
            progress := TRUE;
            state1 := state0;

            state1.dvar_M_HardwareMapP_init_err_sen_idx := 9;
            state1.dvar_M_HardwareMapP := elit_init_error;

            state0 := state1;
        END_IF;
    END_IF;

    // Event "tau".
    IF NOT progress THEN
        b1 := (state0.dvar_M_HardwareMapP) = (elit_init_sensor_check);
        b1 := b1 AND (ivar_s_atdrill);
        IF b1 THEN
            progress := TRUE;
            state1 := state0;

            state1.dvar_M_HardwareMapP_init_err_sen_idx := 10;
            state1.dvar_M_HardwareMapP := elit_init_error;

            state0 := state1;
        END_IF;
    END_IF;

    // Event "tau".
    IF NOT progress THEN
        b1 := (state0.dvar_M_HardwareMapP) = (elit_init_sensor_check);
        b1 := b1 AND (ivar_s_atexit);
        IF b1 THEN
            progress := TRUE;
            state1 := state0;

            state1.dvar_M_HardwareMapP_init_err_sen_idx := 11;
            state1.dvar_M_HardwareMapP := elit_init_error;

            state0 := state1;
        END_IF;
    END_IF;

    // Event "tau".
    IF NOT progress THEN
        b1 := (state0.dvar_M_HardwareMapP) = (elit_init_sensor_check);
        b1 := b1 AND (ivar_s_atspare);
        IF b1 THEN
            progress := TRUE;
            state1 := state0;

            state1.dvar_M_HardwareMapP_init_err_sen_idx := 12;
            state1.dvar_M_HardwareMapP := elit_init_error;

            state0 := state1;
        END_IF;
    END_IF;

    // Event "tau".
    IF NOT progress THEN
        b1 := (state0.dvar_M_HardwareMapP) = (elit_init_sensor_check);
        b1 := b1 AND (ivar_s_clamp);
        IF b1 THEN
            progress := TRUE;
            state1 := state0;

            state1.dvar_M_HardwareMapP_init_err_sen_idx := 13;
            state1.dvar_M_HardwareMapP := elit_init_error;

            state0 := state1;
        END_IF;
    END_IF;

    // Event "tau".
    IF NOT progress THEN
        b1 := (state0.dvar_M_HardwareMapP) = (elit_init_sensor_check);
        b1 := b1 AND (ivar_s_test_ok);
        IF b1 THEN
            progress := TRUE;
            state1 := state0;

            state1.dvar_M_HardwareMapP_init_err_sen_idx := 14;
            state1.dvar_M_HardwareMapP := elit_init_error;

            state0 := state1;
        END_IF;
    END_IF;

    // Event "tau".
    IF NOT progress THEN
        b1 := (state0.dvar_M_HardwareMapP) = (elit_init_sensor_check);
        b1 := b1 AND (NOT(ivar_s_drill_up));
        IF b1 THEN
            progress := TRUE;
            state1 := state0;

            state1.dvar_M_HardwareMapP_init_err_sen_idx := 15;
            state1.dvar_M_HardwareMapP := elit_init_error;

            state0 := state1;
        END_IF;
    END_IF;

    // Event "tau".
    IF NOT progress THEN
        b1 := (state0.dvar_M_HardwareMapP) = (elit_init_sensor_check);
        b1 := b1 AND (ivar_s_drill_down);
        IF b1 THEN
            progress := TRUE;
            state1 := state0;

            state1.dvar_M_HardwareMapP_init_err_sen_idx := 16;
            state1.dvar_M_HardwareMapP := elit_init_error;

            state0 := state1;
        END_IF;
    END_IF;

    // Event "tau".
    IF NOT progress THEN
        b1 := (state0.dvar_M_HardwareMapP) = (elit_init_sensor_check);
        b1 := b1 AND (NOT(ivar_s_turntable));
        IF b1 THEN
            progress := TRUE;
            state1 := state0;

            state1.dvar_M_HardwareMapP_init_err_sen_idx := 17;
            state1.dvar_M_HardwareMapP := elit_init_error;

            state0 := state1;
        END_IF;
    END_IF;

    // Event "tau".
    IF NOT progress THEN
        b1 := (state0.dvar_M_HardwareMapP) = (elit_init_sensor_check);
        b1 := b1 AND (NOT(ivar_s_Pstartbutton));
        b1 := b1 AND (ivar_s_Pstopbutton);
        b1 := b1 AND (NOT(ivar_s_Pautoswitch));
        b1 := b1 AND (NOT(ivar_s_Presetbutton));
        b1 := b1 AND (NOT(ivar_s_Pin4));
        b1 := b1 AND (NOT(ivar_s_Pin5));
        b1 := b1 AND (NOT(ivar_s_Pin6));
        b1 := b1 AND (NOT(ivar_s_Pin7));
        b1 := b1 AND (NOT(ivar_s_atinput));
        b1 := b1 AND (NOT(ivar_s_attest));
        b1 := b1 AND (NOT(ivar_s_atdrill));
        b1 := b1 AND (NOT(ivar_s_atexit));
        b1 := b1 AND (NOT(ivar_s_atspare));
        b1 := b1 AND (NOT(ivar_s_clamp));
        b1 := b1 AND (NOT(ivar_s_test_ok));
        b1 := b1 AND (ivar_s_drill_up);
        b1 := b1 AND (NOT(ivar_s_drill_down));
        b1 := b1 AND (ivar_s_turntable);
        IF b1 THEN
            progress := TRUE;
            state1 := state0;

            state1.dvar_M_HardwareMapP := elit_init_ok;

            state0 := state1;
        END_IF;
    END_IF;

    // Event "tau".
    IF NOT progress THEN
        b1 := (state0.dvar_M_HardwareMapP) = (elit_init_error);
        b1 := b1 AND ((state0.cvar_M_HardwareMapP_t) >= (0.5));
        b1 := b1 AND ((state0.dvar_M_HardwareMapP_init_err_led_idx) = (0));
        IF b1 THEN
            progress := TRUE;
            state1 := state0;

            state1.cvar_M_HardwareMapP_t := 0.0;
            state1.dvar_M_HardwareMapP_init_err_led_idx := 1;
            state1.dvar_M_HardwareMapP_out_a_PledQ1 := TRUE;
            state1.dvar_M_HardwareMapP_out_a_PledQ2 := FALSE;

            state0 := state1;
        END_IF;
    END_IF;

    // Event "tau".
    IF NOT progress THEN
        b1 := (state0.dvar_M_HardwareMapP) = (elit_init_error);
        b1 := b1 AND ((state0.cvar_M_HardwareMapP_t) >= (0.5));
        b1 := b1 AND ((state0.dvar_M_HardwareMapP_init_err_led_idx) = (1));
        IF b1 THEN
            progress := TRUE;
            state1 := state0;

            state1.cvar_M_HardwareMapP_t := 0.0;
            state1.dvar_M_HardwareMapP_init_err_led_idx := 0;
            state1.dvar_M_HardwareMapP_out_a_PledQ1 := FALSE;
            state1.dvar_M_HardwareMapP_out_a_PledQ2 := TRUE;

            state0 := state1;
        END_IF;
    END_IF;

    // Event "tau".
    IF NOT progress THEN
        IF (state0.dvar_M_HardwareMapP) = (elit_init_ok) THEN
            progress := TRUE;
            state1 := state0;

            state1.dvar_M_HardwareMapP_out_a_PledQ1 := FALSE;
            state1.dvar_M_HardwareMapP_out_a_PledQ2 := FALSE;
            state1.dvar_M_HardwareMapP := elit_initialized;

            state0 := state1;
        END_IF;
    END_IF;

    // Event "tau".
    IF NOT progress THEN
        b1 := (state0.dvar_M_HardwareMapP) = (elit_initialized);
        b1 := b1 AND ((state0.dvar_M_HardwareMapP_out_a_Pstartled) <> (FALSE));
        IF b1 THEN
            progress := TRUE;
            state1 := state0;

            state1.dvar_M_HardwareMapP_out_a_Pstartled := FALSE;

            state0 := state1;
        END_IF;
    END_IF;

    // Event "tau".
    IF NOT progress THEN
        b1 := (state0.dvar_M_HardwareMapP) = (elit_initialized);
        b1 := b1 AND ((state0.dvar_M_HardwareMapP_out_a_Presetled) <> (FALSE));
        IF b1 THEN
            progress := TRUE;
            state1 := state0;

            state1.dvar_M_HardwareMapP_out_a_Presetled := FALSE;

            state0 := state1;
        END_IF;
    END_IF;

    // Event "tau".
    IF NOT progress THEN
        b1 := (state0.dvar_M_HardwareMapP) = (elit_initialized);
        b1 := b1 AND ((state0.dvar_M_HardwareMapP_out_a_PledQ1) <> (FALSE));
        IF b1 THEN
            progress := TRUE;
            state1 := state0;

            state1.dvar_M_HardwareMapP_out_a_PledQ1 := FALSE;

            state0 := state1;
        END_IF;
    END_IF;

    // Event "tau".
    IF NOT progress THEN
        b1 := (state0.dvar_M_HardwareMapP) = (elit_initialized);
        b1 := b1 AND ((state0.dvar_M_HardwareMapP_out_a_PledQ2) <> (FALSE));
        IF b1 THEN
            progress := TRUE;
            state1 := state0;

            state1.dvar_M_HardwareMapP_out_a_PledQ2 := FALSE;

            state0 := state1;
        END_IF;
    END_IF;

    // Event "tau".
    IF NOT progress THEN
        b1 := (state0.dvar_M_HardwareMapP) = (elit_initialized);
        b1 := b1 AND ((state0.dvar_M_HardwareMapP_out_a_Pout4) <> (FALSE));
        IF b1 THEN
            progress := TRUE;
            state1 := state0;

            state1.dvar_M_HardwareMapP_out_a_Pout4 := FALSE;

            state0 := state1;
        END_IF;
    END_IF;

    // Event "tau".
    IF NOT progress THEN
        b1 := (state0.dvar_M_HardwareMapP) = (elit_initialized);
        b1 := b1 AND ((state0.dvar_M_HardwareMapP_out_a_Pout5) <> (FALSE));
        IF b1 THEN
            progress := TRUE;
            state1 := state0;

            state1.dvar_M_HardwareMapP_out_a_Pout5 := FALSE;

            state0 := state1;
        END_IF;
    END_IF;

    // Event "tau".
    IF NOT progress THEN
        b1 := (state0.dvar_M_HardwareMapP) = (elit_initialized);
        b1 := b1 AND ((state0.dvar_M_HardwareMapP_out_a_Pout6) <> (FALSE));
        IF b1 THEN
            progress := TRUE;
            state1 := state0;

            state1.dvar_M_HardwareMapP_out_a_Pout6 := FALSE;

            state0 := state1;
        END_IF;
    END_IF;

    // Event "tau".
    IF NOT progress THEN
        b1 := (state0.dvar_M_HardwareMapP) = (elit_initialized);
        b1 := b1 AND ((state0.dvar_M_HardwareMapP_out_a_Pout7) <> (FALSE));
        IF b1 THEN
            progress := TRUE;
            state1 := state0;

            state1.dvar_M_HardwareMapP_out_a_Pout7 := FALSE;

            state0 := state1;
        END_IF;
    END_IF;

    // Event "tau".
    IF NOT progress THEN
        b1 := (state0.dvar_M_HardwareMapP) = (elit_initialized);
        b1 := b1 AND ((state0.dvar_M_HardwareMapP_out_a_drill) <> ((state0.dvar_M_sup_A_drill) = (elit_On)));
        IF b1 THEN
            progress := TRUE;
            state1 := state0;

            state1.dvar_M_HardwareMapP_out_a_drill := (state0.dvar_M_sup_A_drill) = (elit_On);

            state0 := state1;
        END_IF;
    END_IF;

    // Event "tau".
    IF NOT progress THEN
        b1 := (state0.dvar_M_HardwareMapP) = (elit_initialized);
        b1 := b1 AND ((state0.dvar_M_HardwareMapP_out_a_turntable) <> ((state0.dvar_M_sup_A_turntable) = (elit_On)));
        IF b1 THEN
            progress := TRUE;
            state1 := state0;

            state1.dvar_M_HardwareMapP_out_a_turntable := (state0.dvar_M_sup_A_turntable) = (elit_On);

            state0 := state1;
        END_IF;
    END_IF;

    // Event "tau".
    IF NOT progress THEN
        b1 := (state0.dvar_M_HardwareMapP) = (elit_initialized);
        b1 := b1 AND ((state0.dvar_M_HardwareMapP_out_a_drilldown) <> ((state0.dvar_M_sup_A_drilldown) = (elit_On)));
        IF b1 THEN
            progress := TRUE;
            state1 := state0;

            state1.dvar_M_HardwareMapP_out_a_drilldown := (state0.dvar_M_sup_A_drilldown) = (elit_On);

            state0 := state1;
        END_IF;
    END_IF;

    // Event "tau".
    IF NOT progress THEN
        b1 := (state0.dvar_M_HardwareMapP) = (elit_initialized);
        b1 := b1 AND ((state0.dvar_M_HardwareMapP_out_a_drillup) <> ((state0.dvar_M_sup_A_drillup) = (elit_On)));
        IF b1 THEN
            progress := TRUE;
            state1 := state0;

            state1.dvar_M_HardwareMapP_out_a_drillup := (state0.dvar_M_sup_A_drillup) = (elit_On);

            state0 := state1;
        END_IF;
    END_IF;

    // Event "tau".
    IF NOT progress THEN
        b1 := (state0.dvar_M_HardwareMapP) = (elit_initialized);
        b1 := b1 AND ((state0.dvar_M_HardwareMapP_out_a_clamp) <> ((state0.dvar_M_sup_A_clamp) = (elit_On)));
        IF b1 THEN
            progress := TRUE;
            state1 := state0;

            state1.dvar_M_HardwareMapP_out_a_clamp := (state0.dvar_M_sup_A_clamp) = (elit_On);

            state0 := state1;
        END_IF;
    END_IF;

    // Event "tau".
    IF NOT progress THEN
        b1 := (state0.dvar_M_HardwareMapP) = (elit_initialized);
        b1 := b1 AND ((state0.dvar_M_HardwareMapP_out_a_tester) <> ((state0.dvar_M_sup_A_tester) = (elit_On)));
        IF b1 THEN
            progress := TRUE;
            state1 := state0;

            state1.dvar_M_HardwareMapP_out_a_tester := (state0.dvar_M_sup_A_tester) = (elit_On);

            state0 := state1;
        END_IF;
    END_IF;

    // Event "tau".
    IF NOT progress THEN
        b1 := (state0.dvar_M_HardwareMapP) = (elit_initialized);
        b1 := b1 AND ((state0.dvar_M_HardwareMapP_out_a_eject) <> ((state0.dvar_M_sup_A_eject) = (elit_On)));
        IF b1 THEN
            progress := TRUE;
            state1 := state0;

            state1.dvar_M_HardwareMapP_out_a_eject := (state0.dvar_M_sup_A_eject) = (elit_On);

            state0 := state1;
        END_IF;
    END_IF;

    // Event "tau".
    IF NOT progress THEN
        b1 := (state0.dvar_M_HardwareMapP) = (elit_initialized);
        b1 := b1 AND ((state0.dvar_M_HardwareMapP_out_a_processingready) <> ((state0.dvar_M_sup_A_processingready) = (elit_On)));
        IF b1 THEN
            progress := TRUE;
            state1 := state0;

            state1.dvar_M_HardwareMapP_out_a_processingready := (state0.dvar_M_sup_A_processingready) = (elit_On);

            state0 := state1;
        END_IF;
    END_IF;

    // Event "tau".
    IF NOT progress THEN
        b1 := (state0.dvar_M_HardwareMapS) = (elit_init0);
        b1 := b1 AND ((state0.cvar_M_HardwareMapS_t) >= (2.0));
        IF b1 THEN
            progress := TRUE;
            state1 := state0;

            state1.dvar_M_HardwareMapS := elit_init1;

            state0 := state1;
        END_IF;
    END_IF;

    // Event "tau".
    IF NOT progress THEN
        IF (state0.dvar_M_HardwareMapS) = (elit_init1) THEN
            progress := TRUE;
            state1 := state0;

            state1.dvar_M_HardwareMapS_out_a_stopperretract := TRUE;
            state1.dvar_M_HardwareMapS_out_a_conveyer := TRUE;
            state1.cvar_M_HardwareMapS_t := 0.0;
            state1.dvar_M_HardwareMapS := elit_init2;

            state0 := state1;
        END_IF;
    END_IF;

    // Event "tau".
    IF NOT progress THEN
        b1 := (state0.dvar_M_HardwareMapS) = (elit_init2);
        b1 := b1 AND ((state0.cvar_M_HardwareMapS_t) >= (5));
        IF b1 THEN
            progress := TRUE;
            state1 := state0;

            state1.dvar_M_HardwareMapS_out_a_stopperretract := FALSE;
            state1.dvar_M_HardwareMapS_out_a_conveyer := FALSE;
            state1.dvar_M_HardwareMapS := elit_init_sensor_check;

            state0 := state1;
        END_IF;
    END_IF;

    // Event "tau".
    IF NOT progress THEN
        b1 := (state0.dvar_M_HardwareMapS) = (elit_init_sensor_check);
        b1 := b1 AND (ivar_s_Sstartbutton);
        IF b1 THEN
            progress := TRUE;
            state1 := state0;

            state1.dvar_M_HardwareMapS_init_err_sen_idx := 0;
            state1.dvar_M_HardwareMapS := elit_init_error;

            state0 := state1;
        END_IF;
    END_IF;

    // Event "tau".
    IF NOT progress THEN
        b1 := (state0.dvar_M_HardwareMapS) = (elit_init_sensor_check);
        b1 := b1 AND (NOT(ivar_s_Sstopbutton));
        IF b1 THEN
            progress := TRUE;
            state1 := state0;

            state1.dvar_M_HardwareMapS_init_err_sen_idx := 1;
            state1.dvar_M_HardwareMapS := elit_init_error;

            state0 := state1;
        END_IF;
    END_IF;

    // Event "tau".
    IF NOT progress THEN
        b1 := (state0.dvar_M_HardwareMapS) = (elit_init_sensor_check);
        b1 := b1 AND (ivar_s_Sautoswitch);
        IF b1 THEN
            progress := TRUE;
            state1 := state0;

            state1.dvar_M_HardwareMapS_init_err_sen_idx := 2;
            state1.dvar_M_HardwareMapS := elit_init_error;

            state0 := state1;
        END_IF;
    END_IF;

    // Event "tau".
    IF NOT progress THEN
        b1 := (state0.dvar_M_HardwareMapS) = (elit_init_sensor_check);
        b1 := b1 AND (ivar_s_Sresetbutton);
        IF b1 THEN
            progress := TRUE;
            state1 := state0;

            state1.dvar_M_HardwareMapS_init_err_sen_idx := 3;
            state1.dvar_M_HardwareMapS := elit_init_error;

            state0 := state1;
        END_IF;
    END_IF;

    // Event "tau".
    IF NOT progress THEN
        b1 := (state0.dvar_M_HardwareMapS) = (elit_init_sensor_check);
        b1 := b1 AND (ivar_s_Sin4);
        IF b1 THEN
            progress := TRUE;
            state1 := state0;

            state1.dvar_M_HardwareMapS_init_err_sen_idx := 4;
            state1.dvar_M_HardwareMapS := elit_init_error;

            state0 := state1;
        END_IF;
    END_IF;

    // Event "tau".
    IF NOT progress THEN
        b1 := (state0.dvar_M_HardwareMapS) = (elit_init_sensor_check);
        b1 := b1 AND (ivar_s_Sin5);
        IF b1 THEN
            progress := TRUE;
            state1 := state0;

            state1.dvar_M_HardwareMapS_init_err_sen_idx := 5;
            state1.dvar_M_HardwareMapS := elit_init_error;

            state0 := state1;
        END_IF;
    END_IF;

    // Event "tau".
    IF NOT progress THEN
        b1 := (state0.dvar_M_HardwareMapS) = (elit_init_sensor_check);
        b1 := b1 AND (ivar_s_Sin6);
        IF b1 THEN
            progress := TRUE;
            state1 := state0;

            state1.dvar_M_HardwareMapS_init_err_sen_idx := 6;
            state1.dvar_M_HardwareMapS := elit_init_error;

            state0 := state1;
        END_IF;
    END_IF;

    // Event "tau".
    IF NOT progress THEN
        b1 := (state0.dvar_M_HardwareMapS) = (elit_init_sensor_check);
        b1 := b1 AND (ivar_s_Sin7);
        IF b1 THEN
            progress := TRUE;
            state1 := state0;

            state1.dvar_M_HardwareMapS_init_err_sen_idx := 7;
            state1.dvar_M_HardwareMapS := elit_init_error;

            state0 := state1;
        END_IF;
    END_IF;

    // Event "tau".
    IF NOT progress THEN
        b1 := (state0.dvar_M_HardwareMapS) = (elit_init_sensor_check);
        b1 := b1 AND (ivar_s_product);
        IF b1 THEN
            progress := TRUE;
            state1 := state0;

            state1.dvar_M_HardwareMapS_init_err_sen_idx := 8;
            state1.dvar_M_HardwareMapS := elit_init_error;

            state0 := state1;
        END_IF;
    END_IF;

    // Event "tau".
    IF NOT progress THEN
        b1 := (state0.dvar_M_HardwareMapS) = (elit_init_sensor_check);
        b1 := b1 AND (ivar_s_inductive);
        IF b1 THEN
            progress := TRUE;
            state1 := state0;

            state1.dvar_M_HardwareMapS_init_err_sen_idx := 9;
            state1.dvar_M_HardwareMapS := elit_init_error;

            state0 := state1;
        END_IF;
    END_IF;

    // Event "tau".
    IF NOT progress THEN
        b1 := (state0.dvar_M_HardwareMapS) = (elit_init_sensor_check);
        b1 := b1 AND (ivar_s_optical);
        IF b1 THEN
            progress := TRUE;
            state1 := state0;

            state1.dvar_M_HardwareMapS_init_err_sen_idx := 10;
            state1.dvar_M_HardwareMapS := elit_init_error;

            state0 := state1;
        END_IF;
    END_IF;

    // Event "tau".
    IF NOT progress THEN
        b1 := (state0.dvar_M_HardwareMapS) = (elit_init_sensor_check);
        b1 := b1 AND (ivar_s_slidefull);
        IF b1 THEN
            progress := TRUE;
            state1 := state0;

            state1.dvar_M_HardwareMapS_init_err_sen_idx := 11;
            state1.dvar_M_HardwareMapS := elit_init_error;

            state0 := state1;
        END_IF;
    END_IF;

    // Event "tau".
    IF NOT progress THEN
        b1 := (state0.dvar_M_HardwareMapS) = (elit_init_sensor_check);
        b1 := b1 AND (NOT(ivar_s_gate1_opened));
        IF b1 THEN
            progress := TRUE;
            state1 := state0;

            state1.dvar_M_HardwareMapS_init_err_sen_idx := 12;
            state1.dvar_M_HardwareMapS := elit_init_error;

            state0 := state1;
        END_IF;
    END_IF;

    // Event "tau".
    IF NOT progress THEN
        b1 := (state0.dvar_M_HardwareMapS) = (elit_init_sensor_check);
        b1 := b1 AND (ivar_s_gate1_closed);
        IF b1 THEN
            progress := TRUE;
            state1 := state0;

            state1.dvar_M_HardwareMapS_init_err_sen_idx := 13;
            state1.dvar_M_HardwareMapS := elit_init_error;

            state0 := state1;
        END_IF;
    END_IF;

    // Event "tau".
    IF NOT progress THEN
        b1 := (state0.dvar_M_HardwareMapS) = (elit_init_sensor_check);
        b1 := b1 AND (NOT(ivar_s_gate2_opened));
        IF b1 THEN
            progress := TRUE;
            state1 := state0;

            state1.dvar_M_HardwareMapS_init_err_sen_idx := 14;
            state1.dvar_M_HardwareMapS := elit_init_error;

            state0 := state1;
        END_IF;
    END_IF;

    // Event "tau".
    IF NOT progress THEN
        b1 := (state0.dvar_M_HardwareMapS) = (elit_init_sensor_check);
        b1 := b1 AND (ivar_s_gate2_closed);
        IF b1 THEN
            progress := TRUE;
            state1 := state0;

            state1.dvar_M_HardwareMapS_init_err_sen_idx := 15;
            state1.dvar_M_HardwareMapS := elit_init_error;

            state0 := state1;
        END_IF;
    END_IF;

    // Event "tau".
    IF NOT progress THEN
        b1 := (state0.dvar_M_HardwareMapS) = (elit_init_sensor_check);
        b1 := b1 AND (NOT(ivar_s_Sstartbutton));
        b1 := b1 AND (ivar_s_Sstopbutton);
        b1 := b1 AND (NOT(ivar_s_Sautoswitch));
        b1 := b1 AND (NOT(ivar_s_Sresetbutton));
        b1 := b1 AND (NOT(ivar_s_Sin4));
        b1 := b1 AND (NOT(ivar_s_Sin5));
        b1 := b1 AND (NOT(ivar_s_Sin6));
        b1 := b1 AND (NOT(ivar_s_Sin7));
        b1 := b1 AND (NOT(ivar_s_product));
        b1 := b1 AND (NOT(ivar_s_inductive));
        b1 := b1 AND (NOT(ivar_s_optical));
        b1 := b1 AND (NOT(ivar_s_slidefull));
        b1 := b1 AND (ivar_s_gate1_opened);
        b1 := b1 AND (NOT(ivar_s_gate1_closed));
        b1 := b1 AND (ivar_s_gate2_opened);
        b1 := b1 AND (NOT(ivar_s_gate2_closed));
        IF b1 THEN
            progress := TRUE;
            state1 := state0;

            state1.dvar_M_HardwareMapS := elit_init_ok;

            state0 := state1;
        END_IF;
    END_IF;

    // Event "tau".
    IF NOT progress THEN
        b1 := (state0.dvar_M_HardwareMapS) = (elit_init_error);
        b1 := b1 AND ((state0.cvar_M_HardwareMapS_t) >= (0.5));
        b1 := b1 AND ((state0.dvar_M_HardwareMapS_init_err_led_idx) = (0));
        IF b1 THEN
            progress := TRUE;
            state1 := state0;

            state1.cvar_M_HardwareMapS_t := 0.0;
            state1.dvar_M_HardwareMapS_init_err_led_idx := 1;
            state1.dvar_M_HardwareMapS_out_a_SledQ1 := TRUE;
            state1.dvar_M_HardwareMapS_out_a_SledQ2 := FALSE;

            state0 := state1;
        END_IF;
    END_IF;

    // Event "tau".
    IF NOT progress THEN
        b1 := (state0.dvar_M_HardwareMapS) = (elit_init_error);
        b1 := b1 AND ((state0.cvar_M_HardwareMapS_t) >= (0.5));
        b1 := b1 AND ((state0.dvar_M_HardwareMapS_init_err_led_idx) = (1));
        IF b1 THEN
            progress := TRUE;
            state1 := state0;

            state1.cvar_M_HardwareMapS_t := 0.0;
            state1.dvar_M_HardwareMapS_init_err_led_idx := 0;
            state1.dvar_M_HardwareMapS_out_a_SledQ1 := FALSE;
            state1.dvar_M_HardwareMapS_out_a_SledQ2 := TRUE;

            state0 := state1;
        END_IF;
    END_IF;

    // Event "tau".
    IF NOT progress THEN
        IF (state0.dvar_M_HardwareMapS) = (elit_init_ok) THEN
            progress := TRUE;
            state1 := state0;

            state1.dvar_M_HardwareMapS_out_a_SledQ1 := FALSE;
            state1.dvar_M_HardwareMapS_out_a_SledQ2 := FALSE;
            state1.dvar_M_HardwareMapS := elit_initialized;

            state0 := state1;
        END_IF;
    END_IF;

    // Event "tau".
    IF NOT progress THEN
        b1 := (state0.dvar_M_HardwareMapS) = (elit_initialized);
        b1 := b1 AND ((state0.dvar_M_HardwareMapS_out_a_Sstartled) <> (FALSE));
        IF b1 THEN
            progress := TRUE;
            state1 := state0;

            state1.dvar_M_HardwareMapS_out_a_Sstartled := FALSE;

            state0 := state1;
        END_IF;
    END_IF;

    // Event "tau".
    IF NOT progress THEN
        b1 := (state0.dvar_M_HardwareMapS) = (elit_initialized);
        b1 := b1 AND ((state0.dvar_M_HardwareMapS_out_a_Sresetled) <> (FALSE));
        IF b1 THEN
            progress := TRUE;
            state1 := state0;

            state1.dvar_M_HardwareMapS_out_a_Sresetled := FALSE;

            state0 := state1;
        END_IF;
    END_IF;

    // Event "tau".
    IF NOT progress THEN
        b1 := (state0.dvar_M_HardwareMapS) = (elit_initialized);
        b1 := b1 AND ((state0.dvar_M_HardwareMapS_out_a_SledQ1) <> (FALSE));
        IF b1 THEN
            progress := TRUE;
            state1 := state0;

            state1.dvar_M_HardwareMapS_out_a_SledQ1 := FALSE;

            state0 := state1;
        END_IF;
    END_IF;

    // Event "tau".
    IF NOT progress THEN
        b1 := (state0.dvar_M_HardwareMapS) = (elit_initialized);
        b1 := b1 AND ((state0.dvar_M_HardwareMapS_out_a_SledQ2) <> (FALSE));
        IF b1 THEN
            progress := TRUE;
            state1 := state0;

            state1.dvar_M_HardwareMapS_out_a_SledQ2 := FALSE;

            state0 := state1;
        END_IF;
    END_IF;

    // Event "tau".
    IF NOT progress THEN
        b1 := (state0.dvar_M_HardwareMapS) = (elit_initialized);
        b1 := b1 AND ((state0.dvar_M_HardwareMapS_out_a_Sout4) <> (FALSE));
        IF b1 THEN
            progress := TRUE;
            state1 := state0;

            state1.dvar_M_HardwareMapS_out_a_Sout4 := FALSE;

            state0 := state1;
        END_IF;
    END_IF;

    // Event "tau".
    IF NOT progress THEN
        b1 := (state0.dvar_M_HardwareMapS) = (elit_initialized);
        b1 := b1 AND ((state0.dvar_M_HardwareMapS_out_a_Sout5) <> (FALSE));
        IF b1 THEN
            progress := TRUE;
            state1 := state0;

            state1.dvar_M_HardwareMapS_out_a_Sout5 := FALSE;

            state0 := state1;
        END_IF;
    END_IF;

    // Event "tau".
    IF NOT progress THEN
        b1 := (state0.dvar_M_HardwareMapS) = (elit_initialized);
        b1 := b1 AND ((state0.dvar_M_HardwareMapS_out_a_Sout6) <> (FALSE));
        IF b1 THEN
            progress := TRUE;
            state1 := state0;

            state1.dvar_M_HardwareMapS_out_a_Sout6 := FALSE;

            state0 := state1;
        END_IF;
    END_IF;

    // Event "tau".
    IF NOT progress THEN
        b1 := (state0.dvar_M_HardwareMapS) = (elit_initialized);
        b1 := b1 AND ((state0.dvar_M_HardwareMapS_out_a_Sout7) <> (FALSE));
        IF b1 THEN
            progress := TRUE;
            state1 := state0;

            state1.dvar_M_HardwareMapS_out_a_Sout7 := FALSE;

            state0 := state1;
        END_IF;
    END_IF;

    // Event "tau".
    IF NOT progress THEN
        b1 := (state0.dvar_M_HardwareMapS) = (elit_initialized);
        b1 := b1 AND ((state0.dvar_M_HardwareMapS_out_a_conveyer) <> ((state0.dvar_M_sup_A_conveyer) = (elit_On)));
        IF b1 THEN
            progress := TRUE;
            state1 := state0;

            state1.dvar_M_HardwareMapS_out_a_conveyer := (state0.dvar_M_sup_A_conveyer) = (elit_On);

            state0 := state1;
        END_IF;
    END_IF;

    // Event "tau".
    IF NOT progress THEN
        b1 := (state0.dvar_M_HardwareMapS) = (elit_initialized);
        b1 := b1 AND ((state0.dvar_M_HardwareMapS_out_a_gate1) <> ((state0.dvar_M_sup_A_gate1) = (elit_On)));
        IF b1 THEN
            progress := TRUE;
            state1 := state0;

            state1.dvar_M_HardwareMapS_out_a_gate1 := (state0.dvar_M_sup_A_gate1) = (elit_On);

            state0 := state1;
        END_IF;
    END_IF;

    // Event "tau".
    IF NOT progress THEN
        b1 := (state0.dvar_M_HardwareMapS) = (elit_initialized);
        b1 := b1 AND ((state0.dvar_M_HardwareMapS_out_a_gate2) <> ((state0.dvar_M_sup_A_gate2) = (elit_On)));
        IF b1 THEN
            progress := TRUE;
            state1 := state0;

            state1.dvar_M_HardwareMapS_out_a_gate2 := (state0.dvar_M_sup_A_gate2) = (elit_On);

            state0 := state1;
        END_IF;
    END_IF;

    // Event "tau".
    IF NOT progress THEN
        b1 := (state0.dvar_M_HardwareMapS) = (elit_initialized);
        b1 := b1 AND ((state0.dvar_M_HardwareMapS_out_a_stopperretract) <> ((state0.dvar_M_sup_A_stopperretract) = (elit_On)));
        IF b1 THEN
            progress := TRUE;
            state1 := state0;

            state1.dvar_M_HardwareMapS_out_a_stopperretract := (state0.dvar_M_sup_A_stopperretract) = (elit_On);

            state0 := state1;
        END_IF;
    END_IF;

    // Event "tau".
    IF NOT progress THEN
        b1 := (state0.dvar_M_HardwareMapS) = (elit_initialized);
        b1 := b1 AND ((state0.dvar_M_HardwareMapS_out_a_sortingready) <> ((state0.dvar_M_sup_A_sortingready) = (elit_On)));
        IF b1 THEN
            progress := TRUE;
            state1 := state0;

            state1.dvar_M_HardwareMapS_out_a_sortingready := (state0.dvar_M_sup_A_sortingready) = (elit_On);

            state0 := state1;
        END_IF;
    END_IF;

    // Event "tau".
    IF NOT progress THEN
        b1 := (state0.dvar_M_HardwareMapTB) = (elit_init0);
        b1 := b1 AND ((state0.cvar_M_HardwareMapTB_t) >= (2.0));
        IF b1 THEN
            progress := TRUE;
            state1 := state0;

            state1.dvar_M_HardwareMapTB := elit_init1;

            state0 := state1;
        END_IF;
    END_IF;

    // Event "tau".
    IF NOT progress THEN
        IF (state0.dvar_M_HardwareMapTB) = (elit_init1) THEN
            progress := TRUE;
            state1 := state0;

            state1.dvar_M_HardwareMapTB_out_a_airslide := TRUE;
            state1.dvar_M_HardwareMapTB_out_a_conveyerB := TRUE;
            state1.cvar_M_HardwareMapTB_t := 0.0;
            state1.dvar_M_HardwareMapTB := elit_init2;

            state0 := state1;
        END_IF;
    END_IF;

    // Event "tau".
    IF NOT progress THEN
        b1 := (state0.dvar_M_HardwareMapTB) = (elit_init2);
        b1 := b1 AND ((state0.cvar_M_HardwareMapTB_t) >= (5));
        IF b1 THEN
            progress := TRUE;
            state1 := state0;

            state1.dvar_M_HardwareMapTB_out_a_airslide := FALSE;
            state1.dvar_M_HardwareMapTB_out_a_conveyerB := FALSE;
            state1.dvar_M_HardwareMapTB := elit_init_sensor_check;

            state0 := state1;
        END_IF;
    END_IF;

    // Event "tau".
    IF NOT progress THEN
        b1 := (state0.dvar_M_HardwareMapTB) = (elit_init_sensor_check);
        b1 := b1 AND (ivar_s_Tstartbutton);
        IF b1 THEN
            progress := TRUE;
            state1 := state0;

            state1.dvar_M_HardwareMapTB_init_err_sen_idx := 0;
            state1.dvar_M_HardwareMapTB := elit_init_error;

            state0 := state1;
        END_IF;
    END_IF;

    // Event "tau".
    IF NOT progress THEN
        b1 := (state0.dvar_M_HardwareMapTB) = (elit_init_sensor_check);
        b1 := b1 AND (NOT(ivar_s_Tstopbutton));
        IF b1 THEN
            progress := TRUE;
            state1 := state0;

            state1.dvar_M_HardwareMapTB_init_err_sen_idx := 1;
            state1.dvar_M_HardwareMapTB := elit_init_error;

            state0 := state1;
        END_IF;
    END_IF;

    // Event "tau".
    IF NOT progress THEN
        b1 := (state0.dvar_M_HardwareMapTB) = (elit_init_sensor_check);
        b1 := b1 AND (ivar_s_Tautoswitch);
        IF b1 THEN
            progress := TRUE;
            state1 := state0;

            state1.dvar_M_HardwareMapTB_init_err_sen_idx := 2;
            state1.dvar_M_HardwareMapTB := elit_init_error;

            state0 := state1;
        END_IF;
    END_IF;

    // Event "tau".
    IF NOT progress THEN
        b1 := (state0.dvar_M_HardwareMapTB) = (elit_init_sensor_check);
        b1 := b1 AND (ivar_s_Tresetbutton);
        IF b1 THEN
            progress := TRUE;
            state1 := state0;

            state1.dvar_M_HardwareMapTB_init_err_sen_idx := 3;
            state1.dvar_M_HardwareMapTB := elit_init_error;

            state0 := state1;
        END_IF;
    END_IF;

    // Event "tau".
    IF NOT progress THEN
        b1 := (state0.dvar_M_HardwareMapTB) = (elit_init_sensor_check);
        b1 := b1 AND (ivar_s_Tin4);
        IF b1 THEN
            progress := TRUE;
            state1 := state0;

            state1.dvar_M_HardwareMapTB_init_err_sen_idx := 4;
            state1.dvar_M_HardwareMapTB := elit_init_error;

            state0 := state1;
        END_IF;
    END_IF;

    // Event "tau".
    IF NOT progress THEN
        b1 := (state0.dvar_M_HardwareMapTB) = (elit_init_sensor_check);
        b1 := b1 AND (ivar_s_Tin5);
        IF b1 THEN
            progress := TRUE;
            state1 := state0;

            state1.dvar_M_HardwareMapTB_init_err_sen_idx := 5;
            state1.dvar_M_HardwareMapTB := elit_init_error;

            state0 := state1;
        END_IF;
    END_IF;

    // Event "tau".
    IF NOT progress THEN
        b1 := (state0.dvar_M_HardwareMapTB) = (elit_init_sensor_check);
        b1 := b1 AND (ivar_s_Tin6);
        IF b1 THEN
            progress := TRUE;
            state1 := state0;

            state1.dvar_M_HardwareMapTB_init_err_sen_idx := 6;
            state1.dvar_M_HardwareMapTB := elit_init_error;

            state0 := state1;
        END_IF;
    END_IF;

    // Event "tau".
    IF NOT progress THEN
        b1 := (state0.dvar_M_HardwareMapTB) = (elit_init_sensor_check);
        b1 := b1 AND (ivar_s_Tin7);
        IF b1 THEN
            progress := TRUE;
            state1 := state0;

            state1.dvar_M_HardwareMapTB_init_err_sen_idx := 7;
            state1.dvar_M_HardwareMapTB := elit_init_error;

            state0 := state1;
        END_IF;
    END_IF;

    // Event "tau".
    IF NOT progress THEN
        b1 := (state0.dvar_M_HardwareMapTB) = (elit_init_sensor_check);
        b1 := b1 AND (ivar_s_elevator_up);
        IF b1 THEN
            progress := TRUE;
            state1 := state0;

            state1.dvar_M_HardwareMapTB_init_err_sen_idx := 8;
            state1.dvar_M_HardwareMapTB := elit_init_error;

            state0 := state1;
        END_IF;
    END_IF;

    // Event "tau".
    IF NOT progress THEN
        b1 := (state0.dvar_M_HardwareMapTB) = (elit_init_sensor_check);
        b1 := b1 AND (NOT(ivar_s_elevator_down));
        IF b1 THEN
            progress := TRUE;
            state1 := state0;

            state1.dvar_M_HardwareMapTB_init_err_sen_idx := 9;
            state1.dvar_M_HardwareMapTB := elit_init_error;

            state0 := state1;
        END_IF;
    END_IF;

    // Event "tau".
    IF NOT progress THEN
        b1 := (state0.dvar_M_HardwareMapTB) = (elit_init_sensor_check);
        b1 := b1 AND (ivar_s_pusher);
        IF b1 THEN
            progress := TRUE;
            state1 := state0;

            state1.dvar_M_HardwareMapTB_init_err_sen_idx := 10;
            state1.dvar_M_HardwareMapTB := elit_init_error;

            state0 := state1;
        END_IF;
    END_IF;

    // Event "tau".
    IF NOT progress THEN
        b1 := (state0.dvar_M_HardwareMapTB) = (elit_init_sensor_check);
        b1 := b1 AND (ivar_s_opticalT);
        IF b1 THEN
            progress := TRUE;
            state1 := state0;

            state1.dvar_M_HardwareMapTB_init_err_sen_idx := 11;
            state1.dvar_M_HardwareMapTB := elit_init_error;

            state0 := state1;
        END_IF;
    END_IF;

    // Event "tau".
    IF NOT progress THEN
        b1 := (state0.dvar_M_HardwareMapTB) = (elit_init_sensor_check);
        b1 := b1 AND (ivar_s_capacitive);
        IF b1 THEN
            progress := TRUE;
            state1 := state0;

            state1.dvar_M_HardwareMapTB_init_err_sen_idx := 12;
            state1.dvar_M_HardwareMapTB := elit_init_error;

            state0 := state1;
        END_IF;
    END_IF;

    // Event "tau".
    IF NOT progress THEN
        b1 := (state0.dvar_M_HardwareMapTB) = (elit_init_sensor_check);
        b1 := b1 AND (ivar_s_reflective);
        IF b1 THEN
            progress := TRUE;
            state1 := state0;

            state1.dvar_M_HardwareMapTB_init_err_sen_idx := 13;
            state1.dvar_M_HardwareMapTB := elit_init_error;

            state0 := state1;
        END_IF;
    END_IF;

    // Event "tau".
    IF NOT progress THEN
        b1 := (state0.dvar_M_HardwareMapTB) = (elit_init_sensor_check);
        b1 := b1 AND (ivar_s_productheight);
        IF b1 THEN
            progress := TRUE;
            state1 := state0;

            state1.dvar_M_HardwareMapTB_init_err_sen_idx := 14;
            state1.dvar_M_HardwareMapTB := elit_init_error;

            state0 := state1;
        END_IF;
    END_IF;

    // Event "tau".
    IF NOT progress THEN
        b1 := (state0.dvar_M_HardwareMapTB) = (elit_init_sensor_check);
        b1 := b1 AND (ivar_s_Bstartbutton);
        IF b1 THEN
            progress := TRUE;
            state1 := state0;

            state1.dvar_M_HardwareMapTB_init_err_sen_idx := 17;
            state1.dvar_M_HardwareMapTB := elit_init_error;

            state0 := state1;
        END_IF;
    END_IF;

    // Event "tau".
    IF NOT progress THEN
        b1 := (state0.dvar_M_HardwareMapTB) = (elit_init_sensor_check);
        b1 := b1 AND (NOT(ivar_s_Bstopbutton));
        IF b1 THEN
            progress := TRUE;
            state1 := state0;

            state1.dvar_M_HardwareMapTB_init_err_sen_idx := 18;
            state1.dvar_M_HardwareMapTB := elit_init_error;

            state0 := state1;
        END_IF;
    END_IF;

    // Event "tau".
    IF NOT progress THEN
        b1 := (state0.dvar_M_HardwareMapTB) = (elit_init_sensor_check);
        b1 := b1 AND (ivar_s_Bautoswitch);
        IF b1 THEN
            progress := TRUE;
            state1 := state0;

            state1.dvar_M_HardwareMapTB_init_err_sen_idx := 19;
            state1.dvar_M_HardwareMapTB := elit_init_error;

            state0 := state1;
        END_IF;
    END_IF;

    // Event "tau".
    IF NOT progress THEN
        b1 := (state0.dvar_M_HardwareMapTB) = (elit_init_sensor_check);
        b1 := b1 AND (ivar_s_Bresetbutton);
        IF b1 THEN
            progress := TRUE;
            state1 := state0;

            state1.dvar_M_HardwareMapTB_init_err_sen_idx := 20;
            state1.dvar_M_HardwareMapTB := elit_init_error;

            state0 := state1;
        END_IF;
    END_IF;

    // Event "tau".
    IF NOT progress THEN
        b1 := (state0.dvar_M_HardwareMapTB) = (elit_init_sensor_check);
        b1 := b1 AND (ivar_s_Bin4);
        IF b1 THEN
            progress := TRUE;
            state1 := state0;

            state1.dvar_M_HardwareMapTB_init_err_sen_idx := 21;
            state1.dvar_M_HardwareMapTB := elit_init_error;

            state0 := state1;
        END_IF;
    END_IF;

    // Event "tau".
    IF NOT progress THEN
        b1 := (state0.dvar_M_HardwareMapTB) = (elit_init_sensor_check);
        b1 := b1 AND (ivar_s_Bin5);
        IF b1 THEN
            progress := TRUE;
            state1 := state0;

            state1.dvar_M_HardwareMapTB_init_err_sen_idx := 22;
            state1.dvar_M_HardwareMapTB := elit_init_error;

            state0 := state1;
        END_IF;
    END_IF;

    // Event "tau".
    IF NOT progress THEN
        b1 := (state0.dvar_M_HardwareMapTB) = (elit_init_sensor_check);
        b1 := b1 AND (ivar_s_Bin6);
        IF b1 THEN
            progress := TRUE;
            state1 := state0;

            state1.dvar_M_HardwareMapTB_init_err_sen_idx := 23;
            state1.dvar_M_HardwareMapTB := elit_init_error;

            state0 := state1;
        END_IF;
    END_IF;

    // Event "tau".
    IF NOT progress THEN
        b1 := (state0.dvar_M_HardwareMapTB) = (elit_init_sensor_check);
        b1 := b1 AND (ivar_s_Bin7);
        IF b1 THEN
            progress := TRUE;
            state1 := state0;

            state1.dvar_M_HardwareMapTB_init_err_sen_idx := 24;
            state1.dvar_M_HardwareMapTB := elit_init_error;

            state0 := state1;
        END_IF;
    END_IF;

    // Event "tau".
    IF NOT progress THEN
        b1 := (state0.dvar_M_HardwareMapTB) = (elit_init_sensor_check);
        b1 := b1 AND (ivar_s_atin);
        IF b1 THEN
            progress := TRUE;
            state1 := state0;

            state1.dvar_M_HardwareMapTB_init_err_sen_idx := 25;
            state1.dvar_M_HardwareMapTB := elit_init_error;

            state0 := state1;
        END_IF;
    END_IF;

    // Event "tau".
    IF NOT progress THEN
        b1 := (state0.dvar_M_HardwareMapTB) = (elit_init_sensor_check);
        b1 := b1 AND (ivar_s_atseparator);
        IF b1 THEN
            progress := TRUE;
            state1 := state0;

            state1.dvar_M_HardwareMapTB_init_err_sen_idx := 26;
            state1.dvar_M_HardwareMapTB := elit_init_error;

            state0 := state1;
        END_IF;
    END_IF;

    // Event "tau".
    IF NOT progress THEN
        b1 := (state0.dvar_M_HardwareMapTB) = (elit_init_sensor_check);
        b1 := b1 AND (ivar_s_atend);
        IF b1 THEN
            progress := TRUE;
            state1 := state0;

            state1.dvar_M_HardwareMapTB_init_err_sen_idx := 27;
            state1.dvar_M_HardwareMapTB := elit_init_error;

            state0 := state1;
        END_IF;
    END_IF;

    // Event "tau".
    IF NOT progress THEN
        b1 := (state0.dvar_M_HardwareMapTB) = (elit_init_sensor_check);
        b1 := b1 AND (ivar_s_separator_opened);
        IF b1 THEN
            progress := TRUE;
            state1 := state0;

            state1.dvar_M_HardwareMapTB_init_err_sen_idx := 28;
            state1.dvar_M_HardwareMapTB := elit_init_error;

            state0 := state1;
        END_IF;
    END_IF;

    // Event "tau".
    IF NOT progress THEN
        b1 := (state0.dvar_M_HardwareMapTB) = (elit_init_sensor_check);
        b1 := b1 AND (NOT(ivar_s_separator_closed));
        IF b1 THEN
            progress := TRUE;
            state1 := state0;

            state1.dvar_M_HardwareMapTB_init_err_sen_idx := 29;
            state1.dvar_M_HardwareMapTB := elit_init_error;

            state0 := state1;
        END_IF;
    END_IF;

    // Event "tau".
    IF NOT progress THEN
        b1 := (state0.dvar_M_HardwareMapTB) = (elit_init_sensor_check);
        b1 := b1 AND (NOT(ivar_s_Tstartbutton));
        b1 := b1 AND (ivar_s_Tstopbutton);
        b1 := b1 AND (NOT(ivar_s_Tautoswitch));
        b1 := b1 AND (NOT(ivar_s_Tresetbutton));
        b1 := b1 AND (NOT(ivar_s_Tin4));
        b1 := b1 AND (NOT(ivar_s_Tin5));
        b1 := b1 AND (NOT(ivar_s_Tin6));
        b1 := b1 AND (NOT(ivar_s_Tin7));
        b1 := b1 AND (NOT(ivar_s_elevator_up));
        b1 := b1 AND (ivar_s_elevator_down);
        b1 := b1 AND (NOT(ivar_s_pusher));
        b1 := b1 AND (NOT(ivar_s_opticalT));
        b1 := b1 AND (NOT(ivar_s_capacitive));
        b1 := b1 AND (NOT(ivar_s_reflective));
        b1 := b1 AND (NOT(ivar_s_productheight));
        b1 := b1 AND (NOT(ivar_s_Bstartbutton));
        b1 := b1 AND (ivar_s_Bstopbutton);
        b1 := b1 AND (NOT(ivar_s_Bautoswitch));
        b1 := b1 AND (NOT(ivar_s_Bresetbutton));
        b1 := b1 AND (NOT(ivar_s_Bin4));
        b1 := b1 AND (NOT(ivar_s_Bin5));
        b1 := b1 AND (NOT(ivar_s_Bin6));
        b1 := b1 AND (NOT(ivar_s_Bin7));
        b1 := b1 AND (NOT(ivar_s_atin));
        b1 := b1 AND (NOT(ivar_s_atseparator));
        b1 := b1 AND (NOT(ivar_s_atend));
        b1 := b1 AND (NOT(ivar_s_separator_opened));
        b1 := b1 AND (ivar_s_separator_closed);
        IF b1 THEN
            progress := TRUE;
            state1 := state0;

            state1.dvar_M_HardwareMapTB := elit_init_ok;

            state0 := state1;
        END_IF;
    END_IF;

    // Event "tau".
    IF NOT progress THEN
        b1 := (state0.dvar_M_HardwareMapTB) = (elit_init_error);
        b1 := b1 AND ((state0.cvar_M_HardwareMapTB_t) >= (0.5));
        b1 := b1 AND ((state0.dvar_M_HardwareMapTB_init_err_led_idx) = (0));
        IF b1 THEN
            progress := TRUE;
            state1 := state0;

            state1.cvar_M_HardwareMapTB_t := 0.0;
            state1.dvar_M_HardwareMapTB_init_err_led_idx := 1;
            state1.dvar_M_HardwareMapTB_out_a_TledQ1 := TRUE;
            state1.dvar_M_HardwareMapTB_out_a_TledQ2 := FALSE;
            state1.dvar_M_HardwareMapTB_out_a_BledQ1 := TRUE;
            state1.dvar_M_HardwareMapTB_out_a_BledQ2 := FALSE;

            state0 := state1;
        END_IF;
    END_IF;

    // Event "tau".
    IF NOT progress THEN
        b1 := (state0.dvar_M_HardwareMapTB) = (elit_init_error);
        b1 := b1 AND ((state0.cvar_M_HardwareMapTB_t) >= (0.5));
        b1 := b1 AND ((state0.dvar_M_HardwareMapTB_init_err_led_idx) = (1));
        IF b1 THEN
            progress := TRUE;
            state1 := state0;

            state1.cvar_M_HardwareMapTB_t := 0.0;
            state1.dvar_M_HardwareMapTB_init_err_led_idx := 0;
            state1.dvar_M_HardwareMapTB_out_a_TledQ1 := FALSE;
            state1.dvar_M_HardwareMapTB_out_a_TledQ2 := TRUE;
            state1.dvar_M_HardwareMapTB_out_a_BledQ1 := FALSE;
            state1.dvar_M_HardwareMapTB_out_a_BledQ2 := TRUE;

            state0 := state1;
        END_IF;
    END_IF;

    // Event "tau".
    IF NOT progress THEN
        IF (state0.dvar_M_HardwareMapTB) = (elit_init_ok) THEN
            progress := TRUE;
            state1 := state0;

            state1.dvar_M_HardwareMapTB_out_a_TledQ1 := FALSE;
            state1.dvar_M_HardwareMapTB_out_a_TledQ2 := FALSE;
            state1.dvar_M_HardwareMapTB_out_a_BledQ1 := FALSE;
            state1.dvar_M_HardwareMapTB_out_a_BledQ2 := FALSE;
            state1.dvar_M_HardwareMapTB := elit_initialized;

            state0 := state1;
        END_IF;
    END_IF;

    // Event "tau".
    IF NOT progress THEN
        b1 := (state0.dvar_M_HardwareMapTB) = (elit_initialized);
        b1 := b1 AND ((state0.dvar_M_HardwareMapTB_out_a_Tstartled) <> (FALSE));
        IF b1 THEN
            progress := TRUE;
            state1 := state0;

            state1.dvar_M_HardwareMapTB_out_a_Tstartled := FALSE;

            state0 := state1;
        END_IF;
    END_IF;

    // Event "tau".
    IF NOT progress THEN
        b1 := (state0.dvar_M_HardwareMapTB) = (elit_initialized);
        b1 := b1 AND ((state0.dvar_M_HardwareMapTB_out_a_Tresetled) <> (FALSE));
        IF b1 THEN
            progress := TRUE;
            state1 := state0;

            state1.dvar_M_HardwareMapTB_out_a_Tresetled := FALSE;

            state0 := state1;
        END_IF;
    END_IF;

    // Event "tau".
    IF NOT progress THEN
        b1 := (state0.dvar_M_HardwareMapTB) = (elit_initialized);
        b1 := b1 AND ((state0.dvar_M_HardwareMapTB_out_a_TledQ1) <> (FALSE));
        IF b1 THEN
            progress := TRUE;
            state1 := state0;

            state1.dvar_M_HardwareMapTB_out_a_TledQ1 := FALSE;

            state0 := state1;
        END_IF;
    END_IF;

    // Event "tau".
    IF NOT progress THEN
        b1 := (state0.dvar_M_HardwareMapTB) = (elit_initialized);
        b1 := b1 AND ((state0.dvar_M_HardwareMapTB_out_a_TledQ2) <> (FALSE));
        IF b1 THEN
            progress := TRUE;
            state1 := state0;

            state1.dvar_M_HardwareMapTB_out_a_TledQ2 := FALSE;

            state0 := state1;
        END_IF;
    END_IF;

    // Event "tau".
    IF NOT progress THEN
        b1 := (state0.dvar_M_HardwareMapTB) = (elit_initialized);
        b1 := b1 AND ((state0.dvar_M_HardwareMapTB_out_a_Tout4) <> (FALSE));
        IF b1 THEN
            progress := TRUE;
            state1 := state0;

            state1.dvar_M_HardwareMapTB_out_a_Tout4 := FALSE;

            state0 := state1;
        END_IF;
    END_IF;

    // Event "tau".
    IF NOT progress THEN
        b1 := (state0.dvar_M_HardwareMapTB) = (elit_initialized);
        b1 := b1 AND ((state0.dvar_M_HardwareMapTB_out_a_Tout5) <> (FALSE));
        IF b1 THEN
            progress := TRUE;
            state1 := state0;

            state1.dvar_M_HardwareMapTB_out_a_Tout5 := FALSE;

            state0 := state1;
        END_IF;
    END_IF;

    // Event "tau".
    IF NOT progress THEN
        b1 := (state0.dvar_M_HardwareMapTB) = (elit_initialized);
        b1 := b1 AND ((state0.dvar_M_HardwareMapTB_out_a_Tout6) <> (FALSE));
        IF b1 THEN
            progress := TRUE;
            state1 := state0;

            state1.dvar_M_HardwareMapTB_out_a_Tout6 := FALSE;

            state0 := state1;
        END_IF;
    END_IF;

    // Event "tau".
    IF NOT progress THEN
        b1 := (state0.dvar_M_HardwareMapTB) = (elit_initialized);
        b1 := b1 AND ((state0.dvar_M_HardwareMapTB_out_a_Tout7) <> (FALSE));
        IF b1 THEN
            progress := TRUE;
            state1 := state0;

            state1.dvar_M_HardwareMapTB_out_a_Tout7 := FALSE;

            state0 := state1;
        END_IF;
    END_IF;

    // Event "tau".
    IF NOT progress THEN
        b1 := (state0.dvar_M_HardwareMapTB) = (elit_initialized);
        b1 := b1 AND ((state0.dvar_M_HardwareMapTB_out_a_elevator_up) <> ((state0.dvar_M_sup_A_elevator_up) = (elit_On)));
        IF b1 THEN
            progress := TRUE;
            state1 := state0;

            state1.dvar_M_HardwareMapTB_out_a_elevator_up := (state0.dvar_M_sup_A_elevator_up) = (elit_On);

            state0 := state1;
        END_IF;
    END_IF;

    // Event "tau".
    IF NOT progress THEN
        b1 := (state0.dvar_M_HardwareMapTB) = (elit_initialized);
        b1 := b1 AND ((state0.dvar_M_HardwareMapTB_out_a_elevator_down) <> ((state0.dvar_M_sup_A_elevator_down) = (elit_On)));
        IF b1 THEN
            progress := TRUE;
            state1 := state0;

            state1.dvar_M_HardwareMapTB_out_a_elevator_down := (state0.dvar_M_sup_A_elevator_down) = (elit_On);

            state0 := state1;
        END_IF;
    END_IF;

    // Event "tau".
    IF NOT progress THEN
        b1 := (state0.dvar_M_HardwareMapTB) = (elit_initialized);
        b1 := b1 AND ((state0.dvar_M_HardwareMapTB_out_a_pusher) <> ((state0.dvar_M_sup_A_pusher) = (elit_On)));
        IF b1 THEN
            progress := TRUE;
            state1 := state0;

            state1.dvar_M_HardwareMapTB_out_a_pusher := (state0.dvar_M_sup_A_pusher) = (elit_On);

            state0 := state1;
        END_IF;
    END_IF;

    // Event "tau".
    IF NOT progress THEN
        b1 := (state0.dvar_M_HardwareMapTB) = (elit_initialized);
        b1 := b1 AND ((state0.dvar_M_HardwareMapTB_out_a_airslide) <> ((state0.dvar_M_sup_A_airslide) = (elit_On)));
        IF b1 THEN
            progress := TRUE;
            state1 := state0;

            state1.dvar_M_HardwareMapTB_out_a_airslide := (state0.dvar_M_sup_A_airslide) = (elit_On);

            state0 := state1;
        END_IF;
    END_IF;

    // Event "tau".
    IF NOT progress THEN
        b1 := (state0.dvar_M_HardwareMapTB) = (elit_initialized);
        b1 := b1 AND ((state0.dvar_M_HardwareMapTB_out_a_testingready) <> ((state0.dvar_M_sup_A_testingready) = (elit_On)));
        IF b1 THEN
            progress := TRUE;
            state1 := state0;

            state1.dvar_M_HardwareMapTB_out_a_testingready := (state0.dvar_M_sup_A_testingready) = (elit_On);

            state0 := state1;
        END_IF;
    END_IF;

    // Event "tau".
    IF NOT progress THEN
        b1 := (state0.dvar_M_HardwareMapTB) = (elit_initialized);
        b1 := b1 AND ((state0.dvar_M_HardwareMapTB_out_a_Bstartled) <> (FALSE));
        IF b1 THEN
            progress := TRUE;
            state1 := state0;

            state1.dvar_M_HardwareMapTB_out_a_Bstartled := FALSE;

            state0 := state1;
        END_IF;
    END_IF;

    // Event "tau".
    IF NOT progress THEN
        b1 := (state0.dvar_M_HardwareMapTB) = (elit_initialized);
        b1 := b1 AND ((state0.dvar_M_HardwareMapTB_out_a_Bresetled) <> (FALSE));
        IF b1 THEN
            progress := TRUE;
            state1 := state0;

            state1.dvar_M_HardwareMapTB_out_a_Bresetled := FALSE;

            state0 := state1;
        END_IF;
    END_IF;

    // Event "tau".
    IF NOT progress THEN
        b1 := (state0.dvar_M_HardwareMapTB) = (elit_initialized);
        b1 := b1 AND ((state0.dvar_M_HardwareMapTB_out_a_BledQ1) <> (FALSE));
        IF b1 THEN
            progress := TRUE;
            state1 := state0;

            state1.dvar_M_HardwareMapTB_out_a_BledQ1 := FALSE;

            state0 := state1;
        END_IF;
    END_IF;

    // Event "tau".
    IF NOT progress THEN
        b1 := (state0.dvar_M_HardwareMapTB) = (elit_initialized);
        b1 := b1 AND ((state0.dvar_M_HardwareMapTB_out_a_BledQ2) <> (FALSE));
        IF b1 THEN
            progress := TRUE;
            state1 := state0;

            state1.dvar_M_HardwareMapTB_out_a_BledQ2 := FALSE;

            state0 := state1;
        END_IF;
    END_IF;

    // Event "tau".
    IF NOT progress THEN
        b1 := (state0.dvar_M_HardwareMapTB) = (elit_initialized);
        b1 := b1 AND ((state0.dvar_M_HardwareMapTB_out_a_Bout4) <> (FALSE));
        IF b1 THEN
            progress := TRUE;
            state1 := state0;

            state1.dvar_M_HardwareMapTB_out_a_Bout4 := FALSE;

            state0 := state1;
        END_IF;
    END_IF;

    // Event "tau".
    IF NOT progress THEN
        b1 := (state0.dvar_M_HardwareMapTB) = (elit_initialized);
        b1 := b1 AND ((state0.dvar_M_HardwareMapTB_out_a_Bout5) <> (FALSE));
        IF b1 THEN
            progress := TRUE;
            state1 := state0;

            state1.dvar_M_HardwareMapTB_out_a_Bout5 := FALSE;

            state0 := state1;
        END_IF;
    END_IF;

    // Event "tau".
    IF NOT progress THEN
        b1 := (state0.dvar_M_HardwareMapTB) = (elit_initialized);
        b1 := b1 AND ((state0.dvar_M_HardwareMapTB_out_a_Bout6) <> (FALSE));
        IF b1 THEN
            progress := TRUE;
            state1 := state0;

            state1.dvar_M_HardwareMapTB_out_a_Bout6 := FALSE;

            state0 := state1;
        END_IF;
    END_IF;

    // Event "tau".
    IF NOT progress THEN
        b1 := (state0.dvar_M_HardwareMapTB) = (elit_initialized);
        b1 := b1 AND ((state0.dvar_M_HardwareMapTB_out_a_Bout7) <> (FALSE));
        IF b1 THEN
            progress := TRUE;
            state1 := state0;

            state1.dvar_M_HardwareMapTB_out_a_Bout7 := FALSE;

            state0 := state1;
        END_IF;
    END_IF;

    // Event "tau".
    IF NOT progress THEN
        b1 := (state0.dvar_M_HardwareMapTB) = (elit_initialized);
        b1 := b1 AND ((state0.dvar_M_HardwareMapTB_out_a_separator) <> ((state0.dvar_M_sup_A_separator) = (elit_On)));
        IF b1 THEN
            progress := TRUE;
            state1 := state0;

            state1.dvar_M_HardwareMapTB_out_a_separator := (state0.dvar_M_sup_A_separator) = (elit_On);

            state0 := state1;
        END_IF;
    END_IF;

    // Event "tau".
    IF NOT progress THEN
        b1 := (state0.dvar_M_HardwareMapTB) = (elit_initialized);
        b1 := b1 AND ((state0.dvar_M_HardwareMapTB_out_a_conveyerB) <> ((state0.dvar_M_sup_A_conveyerB) = (elit_On)));
        IF b1 THEN
            progress := TRUE;
            state1 := state0;

            state1.dvar_M_HardwareMapTB_out_a_conveyerB := (state0.dvar_M_sup_A_conveyerB) = (elit_On);

            state0 := state1;
        END_IF;
    END_IF;

    // Event "tau".
    IF NOT progress THEN
        b1 := (state0.dvar_M_HardwareMapTB) = (elit_initialized);
        b1 := b1 AND ((state0.dvar_M_HardwareMapTB_out_a_bufferingready) <> ((state0.dvar_M_sup_A_bufferingready) = (elit_On)));
        IF b1 THEN
            progress := TRUE;
            state1 := state0;

            state1.dvar_M_HardwareMapTB_out_a_bufferingready := (state0.dvar_M_sup_A_bufferingready) = (elit_On);

            state0 := state1;
        END_IF;
    END_IF;

    // Done with events?
    IF NOT progress THEN
        EXIT;
    END_IF;

    // Protect against events that are always enabled.
    loopCount := loopCount + 1;
    IF loopCount >= 100 THEN
        loopsKilled := loopsKilled + 1;
        EXIT;
    END_IF;
END_WHILE;
          
END_PROGRAM

